KUKA KRL program: EPS_2_251455_MH52A_A_20251003061554.src

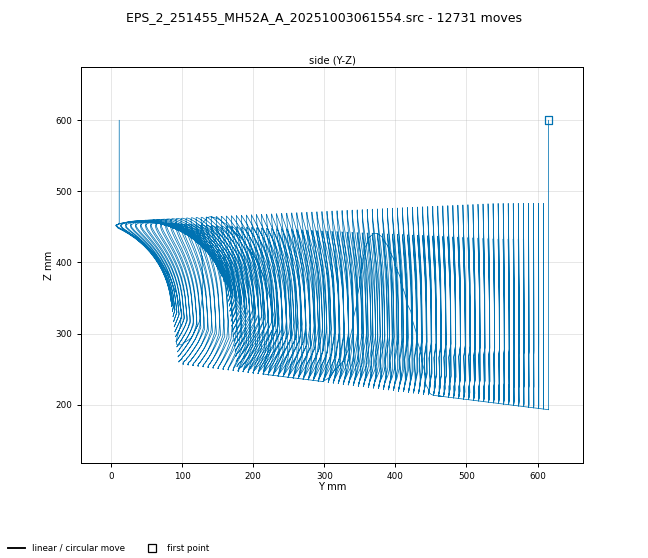
[picture p0: tool path of EPS_2_251455_MH52A_A_20251003061554.src, 12731 of 12733 moves have a stored position in this frame; points joined in program order, loops and branches not executed]
&ACCESS RVP
&REL 4
&COMMENT QRS 19112012
&PARAM EDITMASK = *
DEF PART()
EXT BAS (BAS_COMMAND :IN,REAL :IN )
INT I
BAS (#INITMOV,0 )

;KUKA QRS Post kuka4.cps  Date:22-06-2017 !

File_ID=2878

QRS_PRE_INIT()

;Init var - Until changes are made in qrs_pre_init
Outlet_Square_prg=0
Inlet_1_Square_prg=0
Inlet_2_Square_prg=0
Inlet_3_Square_prg=0
Inlet_4_Square_prg=0
Inlet_5_Square_prg=0

Outlet_1={X 0.000, Y 540.910, Z 382.500, B 0.000, E1 0.000 }
Inlet_1={X 0.000, Y 544.470, Z 332.500, B 0.000, E1 195.000 }
Outlet_1_type=201
Inlet_1_type=201
;QRS#1=Sidecore dimensions
;QRS#2=200-8" PVC SDR 35
;QRS#3=200-8" PVC SDR 35
;QRS#4=
;QRS#5=
;QRS#6=
;QRS#7=
;QRS#8=
;QRS#9=12-08 PSX
;QRS#10=12-08 PSX
;QRS#11=
;QRS#12=
;QRS#13=
;QRS#14=
;QRS#15=
;QRS#16=1220x127x762 2,5'
;QRS#17=EPS Height
;QRS#18=483
;QRS#19=*
;QRS#20= UPDATED VERSION 22-06-2017
;QRS#21=*
Outlet_Square=0100
Inlet_1_Square=0100
Inlet_2_Square=0
Inlet_3_Square=0
Inlet_4_Square=0
Inlet_5_Square=0
Mill_Square=1
Outlet_Square_Prg=204
Inlet_1_Square_prg=204

QRS_INIT()

$ADVANCE=5

; T1
PTP {E1 173.581,E2 173.581}
PTP {X 0,Y 615.464,A -85,B 0,C 180,E1 173.581,E2 173.581,E3 0,E4 0,E5 0,E6 0}
QRS_SPEED_INIT()
LIN {X 0,Y 615.464,Z 600,A -85,B 0,C 180,E1 173.581,E2 173.581,E3 0,E4 0,E5 0,E6 0} C_VEL
LIN {X 0,Y 615.464,Z 202.872,A -85,B 0,C 180,E1 173.581,E2 173.581} C_VEL
LIN {X 0,Y 615.464,Z 194.699,A -85,B 0,C 180,E1 173.581,E2 173.581} C_VEL
LIN {X 0,Y 615.452,Z 192.699,A -85,B 0,C 180,E1 173.395,E2 173.395} C_VEL
LIN {X 0,Y 615.457,Z 192.7,A -85,B 0,C 180,E1 170.801,E2 170.801} C_VEL
LIN {X 0,Y 615.41,Z 192.7,A -85,B 0,C 180,E1 168.138,E2 168.138} C_VEL
LIN {X 0,Y 615.458,Z 192.7,A -85,B 0,C 180,E1 165.45,E2 165.45} C_VEL
LIN {X 0,Y 615.437,Z 192.699,A -85,B 0,C 180,E1 162.728,E2 162.728} C_VEL
LIN {X 0,Y 615.43,Z 192.699,A -85,B 0,C 180,E1 160.66,E2 160.66} C_VEL
LIN {X 0,Y 615.423,Z 192.699,A -85,B 0,C 180,E1 158.566,E2 158.566} C_VEL
LIN {X 0,Y 615.417,Z 192.699,A -85,B 0,C 180,E1 156.441,E2 156.441} C_VEL
LIN {X 0,Y 615.416,Z 192.699,A -85,B 0,C 180,E1 154.281,E2 154.281} C_VEL
LIN {X 0,Y 615.475,Z 192.701,A -85,B 0,C 180,E1 151.54,E2 151.54} C_VEL
LIN {X 0,Y 615.443,Z 192.697,A -85,B 0,C 180,E1 148.91,E2 148.91} C_VEL
LIN {X 0,Y 615.419,Z 192.698,A -85,B 0,C 180,E1 146.465,E2 146.465} C_VEL
LIN {X 0,Y 615.429,Z 192.699,A -85,B 0,C 180,E1 144.165,E2 144.165} C_VEL
LIN {X 0,Y 615.453,Z 192.699,A -85,B 0,C 180,E1 141.929,E2 141.929} C_VEL
LIN {X 0,Y 615.488,Z 192.695,A -85,B 0,C 180,E1 139.394,E2 139.394} C_VEL
LIN {X 0,Y 615.428,Z 192.696,A -85,B 0,C 180,E1 136.75,E2 136.75} C_VEL
LIN {X 0,Y 615.461,Z 192.699,A -85,B 0,C 180,E1 133.995,E2 133.995} C_VEL
LIN {X 0,Y 615.446,Z 192.694,A -85,B 0,C 180,E1 131.09,E2 131.09} C_VEL
LIN {X 0,Y 615.432,Z 192.695,A -85,B 0,C 180,E1 128.903,E2 128.903} C_VEL
LIN {X 0,Y 615.438,Z 192.697,A -85,B 0,C 180,E1 126.423,E2 126.423} C_VEL
LIN {X 0,Y 615.476,Z 192.7,A -85,B 0,C 180,E1 124.018,E2 124.018} C_VEL
LIN {X 0,Y 615.44,Z 192.694,A -85,B 0,C 180,E1 121.079,E2 121.079} C_VEL
LIN {X 0,Y 615.437,Z 192.696,A -85,B 0,C 180,E1 118.656,E2 118.656} C_VEL
LIN {X 0,Y 615.499,Z 192.69,A -85,B 0,C 180,E1 115.711,E2 115.711} C_VEL
LIN {X 0,Y 615.475,Z 192.69,A -85,B 0,C 180,E1 113.553,E2 113.553} C_VEL
LIN {X 0,Y 615.459,Z 192.691,A -85,B 0,C 180,E1 111.43,E2 111.43} C_VEL
LIN {X 0,Y 615.451,Z 192.692,A -85,B 0,C 180,E1 109.336,E2 109.336} C_VEL
LIN {X 0,Y 615.446,Z 192.692,A -85,B 0,C 180,E1 107.269,E2 107.269} C_VEL
LIN {X 0,Y 615.444,Z 192.692,A -85,B 0,C 180,E1 105.225,E2 105.225} C_VEL
LIN {X 0,Y 615.443,Z 192.693,A -85,B 0,C 180,E1 103.2,E2 103.2} C_VEL
LIN {X 0,Y 615.47,Z 192.698,A -85,B 0,C 180,E1 100.525,E2 100.525} C_VEL
LIN {X 0,Y 615.485,Z 192.689,A -85,B 0,C 180,E1 97.874,E2 97.874} C_VEL
LIN {X 0,Y 615.444,Z 192.693,A -85,B 0,C 180,E1 95.24,E2 95.24} C_VEL
LIN {X 0,Y 615.449,Z 192.72,A -85,B 0,C 180,E1 92.985,E2 92.985} C_VEL
LIN {X 0,Y 615.487,Z 207.89,A -85,B 0,C 180,E1 90.326,E2 90.326} C_VEL
LIN {X 0,Y 615.49,Z 222.406,A -85,B 0,C 180,E1 87.811,E2 87.811} C_VEL
LIN {X 0,Y 615.462,Z 329.005,A -85,B 0,C 180,E1 86.542,E2 86.542} C_VEL
LIN {X 0,Y 615.477,Z 341.266,A -85,B 0,C 180,E1 86.276,E2 86.276} C_VEL
LIN {X 0,Y 615.495,Z 353.971,A -85,B 0,C 180,E1 85.866,E2 85.866} C_VEL
LIN {X 0,Y 615.468,Z 366.154,A -85,B 0,C 180,E1 85.333,E2 85.333} C_VEL
LIN {X 0,Y 615.471,Z 377.623,A -85,B 0,C 180,E1 84.676,E2 84.676} C_VEL
LIN {X 0,Y 615.498,Z 387.942,A -85,B 0,C 180,E1 83.937,E2 83.937} C_VEL
LIN {X 0,Y 615.497,Z 397.467,A -85,B 0,C 180,E1 83.098,E2 83.098} C_VEL
LIN {X 0,Y 615.496,Z 406.346,A -85,B 0,C 180,E1 82.124,E2 82.124} C_VEL
LIN {X 0,Y 615.496,Z 413.655,A -85,B 0,C 180,E1 81.132,E2 81.132} C_VEL
LIN {X 0,Y 615.499,Z 419.524,A -85,B 0,C 180,E1 80.138,E2 80.138} C_VEL
LIN {X 0,Y 615.494,Z 424.293,A -85,B 0,C 180,E1 79.108,E2 79.108} C_VEL
LIN {X 0,Y 615.496,Z 427.682,A -85,B 0,C 180,E1 78.139,E2 78.139} C_VEL
LIN {X 0,Y 615.495,Z 429.469,A -85,B 0,C 180,E1 77.47,E2 77.47} C_VEL
LIN {X 0,Y 615.496,Z 430.806,A -85,B 0,C 180,E1 76.799,E2 76.799} C_VEL
LIN {X 0,Y 615.498,Z 431.817,A -85,B 0,C 180,E1 76.063,E2 76.063} C_VEL
LIN {X 0,Y 615.494,Z 432.275,A -85,B 0,C 180,E1 75.451,E2 75.451} C_VEL
LIN {X 0,Y 615.496,Z 432.351,A -85,B 0,C 180,E1 74.774,E2 74.774} C_VEL
LIN {X 0,Y 615.494,Z 431.486,A -85,B 0,C 180,E1 73.566,E2 73.566} C_VEL
LIN {X 0,Y 615.495,Z 430.097,A -85,B 0,C 180,E1 72.73,E2 72.73} C_VEL
LIN {X 0,Y 615.498,Z 428.448,A -85,B 0,C 180,E1 72.044,E2 72.044} C_VEL
LIN {X 0,Y 615.496,Z 425.076,A -85,B 0,C 180,E1 71.009,E2 71.009} C_VEL
LIN {X 0,Y 615.496,Z 420.512,A -85,B 0,C 180,E1 69.968,E2 69.968} C_VEL
LIN {X 0,Y 615.496,Z 414.592,A -85,B 0,C 180,E1 68.92,E2 68.92} C_VEL
LIN {X 0,Y 615.497,Z 406.993,A -85,B 0,C 180,E1 67.865,E2 67.865} C_VEL
LIN {X 0,Y 615.498,Z 399.11,A -85,B 0,C 180,E1 66.979,E2 66.979} C_VEL
LIN {X 0,Y 615.497,Z 389.577,A -85,B 0,C 180,E1 66.103,E2 66.103} C_VEL
LIN {X 0,Y 615.48,Z 379.696,A -85,B 0,C 180,E1 65.37,E2 65.37} C_VEL
LIN {X 0,Y 615.466,Z 368.848,A -85,B 0,C 180,E1 64.72,E2 64.72} C_VEL
LIN {X 0,Y 615.483,Z 356.684,A -85,B 0,C 180,E1 64.149,E2 64.149} C_VEL
LIN {X 0,Y 615.446,Z 345.029,A -85,B 0,C 180,E1 63.738,E2 63.738} C_VEL
LIN {X 0,Y 615.434,Z 332.142,A -85,B 0,C 180,E1 63.425,E2 63.425} C_VEL
LIN {X 0,Y 615.438,Z 314.635,A -85,B 0,C 180,E1 63.184,E2 63.184} C_VEL
LIN {X 0,Y 615.475,Z 222.334,A -85,B 0,C 180,E1 62.086,E2 62.086} C_VEL
LIN {X 0,Y 615.486,Z 206.099,A -85,B 0,C 180,E1 59.272,E2 59.272} C_VEL
LIN {X 0,Y 615.471,Z 192.69,A -85,B 0,C 180,E1 56.911,E2 56.911} C_VEL
LIN {X 0,Y 615.487,Z 192.686,A -85,B 0,C 180,E1 54.166,E2 54.166} C_VEL
LIN {X 0,Y 615.486,Z 192.692,A -85,B 0,C 180,E1 51.934,E2 51.934} C_VEL
LIN {X 0,Y 615.477,Z 192.696,A -85,B 0,C 180,E1 49.396,E2 49.396} C_VEL
LIN {X 0,Y 615.476,Z 192.685,A -85,B 0,C 180,E1 46.758,E2 46.758} C_VEL
LIN {X 0,Y 615.488,Z 192.695,A -85,B 0,C 180,E1 44.001,E2 44.001} C_VEL
LIN {X 0,Y 615.469,Z 192.695,A -85,B 0,C 180,E1 41.475,E2 41.475} C_VEL
LIN {X 0,Y 615.468,Z 192.687,A -85,B 0,C 180,E1 38.906,E2 38.906} C_VEL
LIN {X 0,Y 615.488,Z 192.688,A -85,B 0,C 180,E1 36.424,E2 36.424} C_VEL
LIN {X 0,Y 615.492,Z 192.701,A -85,B 0,C 180,E1 34.021,E2 34.021} C_VEL
LIN {X 0,Y 615.466,Z 192.696,A -85,B 0,C 180,E1 31.686,E2 31.686} C_VEL
LIN {X 0,Y 615.454,Z 192.692,A -85,B 0,C 180,E1 29.408,E2 29.408} C_VEL
LIN {X 0,Y 615.465,Z 192.688,A -85,B 0,C 180,E1 27.049,E2 27.049} C_VEL
LIN {X 0,Y 615.476,Z 192.698,A -85,B 0,C 180,E1 24.015,E2 24.015} C_VEL
LIN {X 0,Y 615.449,Z 192.692,A -85,B 0,C 180,E1 21.433,E2 21.433} C_VEL
LIN {X 0,Y 615.493,Z 192.692,A -85,B 0,C 180,E1 18.618,E2 18.618} C_VEL
LIN {X 0,Y 615.452,Z 192.696,A -85,B 0,C 180,E1 15.906,E2 15.906} C_VEL
LIN {X 0,Y 615.447,Z 192.696,A -85,B 0,C 180,E1 13.875,E2 13.875} C_VEL
LIN {X 0,Y 615.444,Z 192.695,A -85,B 0,C 180,E1 11.861,E2 11.861} C_VEL
LIN {X 0,Y 615.442,Z 192.695,A -85,B 0,C 180,E1 9.863,E2 9.863} C_VEL
LIN {X 0,Y 615.439,Z 192.695,A -85,B 0,C 180,E1 7.876,E2 7.876} C_VEL
LIN {X 0,Y 615.463,Z 192.691,A -85,B 0,C 180,E1 5.241,E2 5.241} C_VEL
LIN {X 0,Y 615.484,Z 192.701,A -85,B 0,C 180,E1 2.618,E2 2.618} C_VEL
LIN {X 0,Y 615.43,Z 192.697,A -85,B 0,C 180,E1 0,E2 0} C_VEL
LIN {X 0,Y 615.431,Z 192.697,A -85,B 0,C 180,E1 -1.963,E2 -1.963} C_VEL
LIN {X 0,Y 615.429,Z 192.697,A -85,B 0,C 180,E1 -3.929,E2 -3.929} C_VEL
LIN {X 0,Y 615.428,Z 192.697,A -85,B 0,C 180,E1 -5.899,E2 -5.899} C_VEL
LIN {X 0,Y 615.423,Z 192.698,A -85,B 0,C 180,E1 -7.877,E2 -7.877} C_VEL
LIN {X 0,Y 615.424,Z 192.698,A -85,B 0,C 180,E1 -9.863,E2 -9.863} C_VEL
LIN {X 0,Y 615.421,Z 192.698,A -85,B 0,C 180,E1 -11.862,E2 -11.862} C_VEL
LIN {X 0,Y 615.458,Z 192.697,A -85,B 0,C 180,E1 -14.55,E2 -14.55} C_VEL
LIN {X 0,Y 615.445,Z 192.7,A -85,B 0,C 180,E1 -17.272,E2 -17.272} C_VEL
LIN {X 0,Y 615.433,Z 192.7,A -85,B 0,C 180,E1 -19.34,E2 -19.34} C_VEL
LIN {X 0,Y 615.422,Z 192.7,A -85,B 0,C 180,E1 -21.435,E2 -21.435} C_VEL
LIN {X 0,Y 615.411,Z 192.701,A -85,B 0,C 180,E1 -23.56,E2 -23.56} C_VEL
LIN {X 0,Y 615.412,Z 192.7,A -85,B 0,C 180,E1 -25.719,E2 -25.719} C_VEL
LIN {X 0,Y 615.47,Z 192.701,A -85,B 0,C 180,E1 -28.455,E2 -28.455} C_VEL
LIN {X 0,Y 615.443,Z 192.698,A -85,B 0,C 180,E1 -31.086,E2 -31.086} C_VEL
LIN {X 0,Y 615.419,Z 192.698,A -85,B 0,C 180,E1 -33.53,E2 -33.53} C_VEL
LIN {X 0,Y 615.429,Z 192.699,A -85,B 0,C 180,E1 -35.831,E2 -35.831} C_VEL
LIN {X 0,Y 615.454,Z 192.699,A -85,B 0,C 180,E1 -38.071,E2 -38.071} C_VEL
LIN {X 0,Y 615.486,Z 192.695,A -85,B 0,C 180,E1 -40.607,E2 -40.607} C_VEL
LIN {X 0,Y 615.43,Z 192.696,A -85,B 0,C 180,E1 -43.25,E2 -43.25} C_VEL
LIN {X 0,Y 615.467,Z 192.699,A -85,B 0,C 180,E1 -46.005,E2 -46.005} C_VEL
LIN {X 0,Y 615.448,Z 192.693,A -85,B 0,C 180,E1 -48.91,E2 -48.91} C_VEL
LIN {X 0,Y 615.435,Z 192.695,A -85,B 0,C 180,E1 -51.095,E2 -51.095} C_VEL
LIN {X 0,Y 615.444,Z 192.698,A -85,B 0,C 180,E1 -53.575,E2 -53.575} C_VEL
LIN {X 0,Y 615.486,Z 192.689,A -85,B 0,C 180,E1 -56.467,E2 -56.467} C_VEL
LIN {X 0,Y 615.442,Z 192.693,A -85,B 0,C 180,E1 -59.08,E2 -59.08} C_VEL
LIN {X 0,Y 615.458,Z 192.698,A -85,B 0,C 180,E1 -61.555,E2 -61.555} C_VEL
LIN {X 0,Y 615.48,Z 192.688,A -85,B 0,C 180,E1 -64.433,E2 -64.433} C_VEL
LIN {X 0,Y 615.447,Z 192.693,A -85,B 0,C 180,E1 -67.044,E2 -67.044} C_VEL
LIN {X 0,Y 615.482,Z 210.777,A -85,B 0,C 180,E1 -69.445,E2 -69.445} C_VEL
LIN {X 0,Y 615.489,Z 232.021,A -85,B 0,C 180,E1 -72.215,E2 -72.215} C_VEL
LIN {X 0,Y 615.494,Z 253.241,A -85,B 0,C 180,E1 -74.944,E2 -74.944} C_VEL
LIN {X 0,Y 615.452,Z 270.301,A -85,B 0,C 180,E1 -77.113,E2 -77.113} C_VEL
LIN {X 0,Y 615.478,Z 378.828,A -85,B 0,C 180,E1 -78.41,E2 -78.41} C_VEL
LIN {X 0,Y 615.47,Z 391.343,A -85,B 0,C 180,E1 -78.681,E2 -78.681} C_VEL
LIN {X 0,Y 615.486,Z 404.643,A -85,B 0,C 180,E1 -79.114,E2 -79.114} C_VEL
LIN {X 0,Y 615.483,Z 416.474,A -85,B 0,C 180,E1 -79.639,E2 -79.639} C_VEL
LIN {X 0,Y 615.495,Z 427.99,A -85,B 0,C 180,E1 -80.304,E2 -80.304} C_VEL
LIN {X 0,Y 615.499,Z 438.337,A -85,B 0,C 180,E1 -81.05,E2 -81.05} C_VEL
LIN {X 0,Y 615.497,Z 446.807,A -85,B 0,C 180,E1 -81.794,E2 -81.794} C_VEL
LIN {X 0,Y 615.498,Z 454.602,A -85,B 0,C 180,E1 -82.619,E2 -82.619} C_VEL
LIN {X 0,Y 615.496,Z 462.199,A -85,B 0,C 180,E1 -83.607,E2 -83.607} C_VEL
LIN {X 0,Y 615.498,Z 469.201,A -85,B 0,C 180,E1 -84.758,E2 -84.758} C_VEL
LIN {X 0,Y 615.494,Z 473.848,A -85,B 0,C 180,E1 -85.743,E2 -85.743} C_VEL
LIN {X 0,Y 615.494,Z 477.396,A -85,B 0,C 180,E1 -86.726,E2 -86.726} C_VEL
LIN {X 0,Y 615.497,Z 479.231,A -85,B 0,C 180,E1 -87.381,E2 -87.381} C_VEL
LIN {X 0,Y 615.499,Z 480.606,A -85,B 0,C 180,E1 -88.036,E2 -88.036} C_VEL
LIN {X 0,Y 615.496,Z 482.173,A -85,B 0,C 180,E1 -89.345,E2 -89.345} C_VEL
LIN {X 0,Y 615.494,Z 482.389,A -85,B 0,C 180,E1 -89.999,E2 -89.999} C_VEL
LIN {X 0,Y 615.495,Z 481.581,A -85,B 0,C 180,E1 -91.307,E2 -91.307} C_VEL
LIN {X 0,Y 615.499,Z 480.61,A -85,B 0,C 180,E1 -91.962,E2 -91.962} C_VEL
LIN {X 0,Y 615.497,Z 479.236,A -85,B 0,C 180,E1 -92.616,E2 -92.616} C_VEL
LIN {X 0,Y 615.496,Z 476.354,A -85,B 0,C 180,E1 -93.599,E2 -93.599} C_VEL
LIN {X 0,Y 615.498,Z 472.448,A -85,B 0,C 180,E1 -94.583,E2 -94.583} C_VEL
LIN {X 0,Y 615.499,Z 467.414,A -85,B 0,C 180,E1 -95.568,E2 -95.568} C_VEL
LIN {X 0,Y 615.496,Z 460.87,A -85,B 0,C 180,E1 -96.583,E2 -96.583} C_VEL
LIN {X 0,Y 615.497,Z 453.15,A -85,B 0,C 180,E1 -97.544,E2 -97.544} C_VEL
LIN {X 0,Y 615.498,Z 445.065,A -85,B 0,C 180,E1 -98.369,E2 -98.369} C_VEL
LIN {X 0,Y 615.499,Z 435.194,A -85,B 0,C 180,E1 -99.197,E2 -99.197} C_VEL
LIN {X 0,Y 615.492,Z 424.016,A -85,B 0,C 180,E1 -99.943,E2 -99.943} C_VEL
LIN {X 0,Y 615.485,Z 413.067,A -85,B 0,C 180,E1 -100.525,E2 -100.525} C_VEL
LIN {X 0,Y 615.476,Z 400.535,A -85,B 0,C 180,E1 -101.039,E2 -101.039} C_VEL
LIN {X 0,Y 615.471,Z 388.165,A -85,B 0,C 180,E1 -101.4,E2 -101.4} C_VEL
LIN {X 0,Y 615.481,Z 374.629,A -85,B 0,C 180,E1 -101.65,E2 -101.65} C_VEL
LIN {X 0,Y 615.452,Z 270.319,A -85,B 0,C 180,E1 -102.885,E2 -102.885} C_VEL
LIN {X 0,Y 615.487,Z 249.28,A -85,B 0,C 180,E1 -105.563,E2 -105.563} C_VEL
LIN {X 0,Y 615.456,Z 227.019,A -85,B 0,C 180,E1 -108.434,E2 -108.434} C_VEL
LIN {X 0,Y 615.482,Z 206.806,A -85,B 0,C 180,E1 -111.078,E2 -111.078} C_VEL
LIN {X 0,Y 615.447,Z 192.693,A -85,B 0,C 180,E1 -112.976,E2 -112.976} C_VEL
LIN {X 0,Y 615.499,Z 192.686,A -85,B 0,C 180,E1 -115.711,E2 -115.711} C_VEL
LIN {X 0,Y 615.451,Z 192.695,A -85,B 0,C 180,E1 -118.656,E2 -118.656} C_VEL
LIN {X 0,Y 615.447,Z 192.692,A -85,B 0,C 180,E1 -121.079,E2 -121.079} C_VEL
LIN {X 0,Y 615.496,Z 192.701,A -85,B 0,C 180,E1 -124.017,E2 -124.017} C_VEL
LIN {X 0,Y 615.454,Z 192.697,A -85,B 0,C 180,E1 -126.422,E2 -126.422} C_VEL
LIN {X 0,Y 615.445,Z 192.692,A -85,B 0,C 180,E1 -129.057,E2 -129.057} C_VEL
LIN {X 0,Y 615.487,Z 192.689,A -85,B 0,C 180,E1 -131.468,E2 -131.468} C_VEL
LIN {X 0,Y 615.465,Z 192.698,A -85,B 0,C 180,E1 -134.145,E2 -134.145} C_VEL
LIN {X 0,Y 615.436,Z 192.694,A -85,B 0,C 180,E1 -136.751,E2 -136.751} C_VEL
LIN {X 0,Y 615.489,Z 192.69,A -85,B 0,C 180,E1 -139.393,E2 -139.393} C_VEL
LIN {X 0,Y 615.467,Z 192.699,A -85,B 0,C 180,E1 -141.982,E2 -141.982} C_VEL
LIN {X 0,Y 615.435,Z 192.696,A -85,B 0,C 180,E1 -144.38,E2 -144.38} C_VEL
LIN {X 0,Y 615.437,Z 192.694,A -85,B 0,C 180,E1 -146.76,E2 -146.76} C_VEL
LIN {X 0,Y 615.465,Z 192.692,A -85,B 0,C 180,E1 -149.079,E2 -149.079} C_VEL
LIN {X 0,Y 615.441,Z 192.697,A -85,B 0,C 180,E1 -152.082,E2 -152.082} C_VEL
LIN {X 0,Y 615.428,Z 192.696,A -85,B 0,C 180,E1 -154.429,E2 -154.429} C_VEL
LIN {X 0,Y 615.484,Z 192.693,A -85,B 0,C 180,E1 -157.155,E2 -157.155} C_VEL
LIN {X 0,Y 615.438,Z 192.698,A -85,B 0,C 180,E1 -159.965,E2 -159.965} C_VEL
LIN {X 0,Y 615.431,Z 192.698,A -85,B 0,C 180,E1 -162.041,E2 -162.041} C_VEL
LIN {X 0,Y 615.425,Z 192.698,A -85,B 0,C 180,E1 -164.093,E2 -164.093} C_VEL
LIN {X 0,Y 615.424,Z 192.698,A -85,B 0,C 180,E1 -166.124,E2 -166.124} C_VEL
LIN {X 0,Y 615.423,Z 192.698,A -85,B 0,C 180,E1 -168.138,E2 -168.138} C_VEL
LIN {X 0,Y 615.419,Z 192.698,A -85,B 0,C 180,E1 -170.137,E2 -170.137} C_VEL
LIN {X 0,Y 615.458,Z 192.696,A -85,B 0,C 180,E1 -172.784,E2 -172.784} C_VEL
LIN {X 0,Y 615.462,Z 192.7,A -85,B 0,C 180,E1 -175.415,E2 -175.415} C_VEL
LIN {X 0,Y 615.417,Z 192.698,A -85,B 0,C 180,E1 -178.036,E2 -178.036} C_VEL
LIN {X 0,Y 615.452,Z 192.698,A -85,B 0,C 180,E1 -180.654,E2 -180.654} C_VEL
LIN {X 0,Y 615.462,Z 192.7,A -85,B 0,C 180,E1 -183.273,E2 -183.273} C_VEL
LIN {X 0,Y 615.412,Z 192.7,A -85,B 0,C 180,E1 -185.899,E2 -185.899} C_VEL
LIN {X 0,Y 615.452,Z 192.699,A -85,B 0,C 180,E1 -186.605,E2 -186.605} C_VEL
LIN {X 0,Y 614.783,Z 192.848,A -85,B 0,C 180,E1 -187.151,E2 -187.151} C_VEL
LIN {X 0,Y 611.954,Z 193.251,A -85,B 0,C 180,E1 -188.037,E2 -188.037} C_VEL
LIN {X 0,Y 609.556,Z 193.564,A -85,B 0,C 180,E1 -188.749,E2 -188.749} C_VEL
LIN {X 0,Y 608.507,Z 193.685,A -85,B 0,C 180,E1 -189.299,E2 -189.299} C_VEL
LIN {X 0,Y 608.411,Z 193.695,A -85,B 0,C 180,E1 -189.485,E2 -189.485} C_VEL
LIN {X 0,Y 608.428,Z 193.694,A -85,B 0,C 180,E1 -191.324,E2 -191.324} C_VEL
LIN {X 0,Y 608.405,Z 193.694,A -85,B 0,C 180,E1 -194.039,E2 -194.039} C_VEL
LIN {X 0,Y 608.437,Z 193.7,A -85,B 0,C 180,E1 -196.784,E2 -196.784} C_VEL
LIN {X 0,Y 608.392,Z 193.695,A -85,B 0,C 180,E1 -199.572,E2 -199.572} C_VEL
LIN {X 0,Y 608.408,Z 193.693,A -85,B 0,C 180,E1 -201.694,E2 -201.694} C_VEL
LIN {X 0,Y 608.416,Z 193.701,A -85,B 0,C 180,E1 -204.572,E2 -204.572} C_VEL
LIN {X 0,Y 608.395,Z 193.695,A -85,B 0,C 180,E1 -207.52,E2 -207.52} C_VEL
LIN {X 0,Y 608.412,Z 193.694,A -85,B 0,C 180,E1 -209.974,E2 -209.974} C_VEL
LIN {X 0,Y 608.451,Z 193.698,A -85,B 0,C 180,E1 -212.531,E2 -212.531} C_VEL
LIN {X 0,Y 608.397,Z 193.695,A -85,B 0,C 180,E1 -215.281,E2 -215.281} C_VEL
LIN {X 0,Y 608.425,Z 193.692,A -85,B 0,C 180,E1 -217.749,E2 -217.749} C_VEL
LIN {X 0,Y 608.441,Z 193.699,A -85,B 0,C 180,E1 -220.336,E2 -220.336} C_VEL
LIN {X 0,Y 608.412,Z 193.694,A -85,B 0,C 180,E1 -222.963,E2 -222.963} C_VEL
LIN {X 0,Y 608.407,Z 193.693,A -85,B 0,C 180,E1 -225.206,E2 -225.206} C_VEL
LIN {X 0,Y 608.434,Z 193.695,A -85,B 0,C 180,E1 -227.943,E2 -227.943} C_VEL
LIN {X 0,Y 608.446,Z 193.691,A -85,B 0,C 180,E1 -230.705,E2 -230.705} C_VEL
LIN {X 0,Y 608.405,Z 193.693,A -85,B 0,C 180,E1 -233.087,E2 -233.087} C_VEL
LIN {X 0,Y 608.43,Z 193.692,A -85,B 0,C 180,E1 -235.533,E2 -235.533} C_VEL
LIN {X 0,Y 608.444,Z 193.696,A -85,B 0,C 180,E1 -237.909,E2 -237.909} C_VEL
LIN {X 0,Y 608.479,Z 193.692,A -85,B 0,C 180,E1 -240.225,E2 -240.225} C_VEL
LIN {X 0,Y 608.407,Z 193.694,A -85,B 0,C 180,E1 -243.228,E2 -243.228} C_VEL
LIN {X 0,Y 608.48,Z 193.693,A -85,B 0,C 180,E1 -245.847,E2 -245.847} C_VEL
LIN {X 0,Y 608.455,Z 193.691,A -85,B 0,C 180,E1 -248.311,E2 -248.311} C_VEL
LIN {X 0,Y 608.429,Z 193.691,A -85,B 0,C 180,E1 -251.133,E2 -251.133} C_VEL
LIN {X 0,Y 608.457,Z 193.696,A -85,B 0,C 180,E1 -253.909,E2 -253.909} C_VEL
LIN {X 0,Y 608.435,Z 193.69,A -85,B 0,C 180,E1 -256.645,E2 -256.645} C_VEL
LIN {X 0,Y 608.441,Z 193.693,A -85,B 0,C 180,E1 -259.352,E2 -259.352} C_VEL
LIN {X 0,Y 608.475,Z 193.689,A -85,B 0,C 180,E1 -262.035,E2 -262.035} C_VEL
LIN {X 0,Y 608.43,Z 193.69,A -85,B 0,C 180,E1 -264.699,E2 -264.699} C_VEL
LIN {X 0,Y 608.44,Z 193.816,A -85,B 0,C 180,E1 -266.98,E2 -266.98} C_VEL
LIN {X 0,Y 608.486,Z 207.153,A -85,B 0,C 180,E1 -269.339,E2 -269.339} C_VEL
LIN {X 0,Y 608.499,Z 222.784,A -85,B 0,C 180,E1 -272.049,E2 -272.049} C_VEL
LIN {X 0,Y 608.52,Z 329.538,A -85,B 0,C 180,E1 -273.332,E2 -273.332} C_VEL
LIN {X 0,Y 608.518,Z 343.159,A -85,B 0,C 180,E1 -273.643,E2 -273.643} C_VEL
LIN {X 0,Y 608.535,Z 355.415,A -85,B 0,C 180,E1 -274.057,E2 -274.057} C_VEL
LIN {X 0,Y 608.474,Z 366.473,A -85,B 0,C 180,E1 -274.555,E2 -274.555} C_VEL
LIN {X 0,Y 608.457,Z 377.952,A -85,B 0,C 180,E1 -275.22,E2 -275.22} C_VEL
LIN {X 0,Y 608.498,Z 388.292,A -85,B 0,C 180,E1 -275.967,E2 -275.967} C_VEL
LIN {X 0,Y 608.46,Z 397.701,A -85,B 0,C 180,E1 -276.8,E2 -276.8} C_VEL
LIN {X 0,Y 608.454,Z 406.781,A -85,B 0,C 180,E1 -277.801,E2 -277.801} C_VEL
LIN {X 0,Y 608.449,Z 414.134,A -85,B 0,C 180,E1 -278.804,E2 -278.804} C_VEL
LIN {X 0,Y 608.433,Z 419.13,A -85,B 0,C 180,E1 -279.642,E2 -279.642} C_VEL
LIN {X 0,Y 608.436,Z 423.991,A -85,B 0,C 180,E1 -280.651,E2 -280.651} C_VEL
LIN {X 0,Y 608.434,Z 427.727,A -85,B 0,C 180,E1 -281.662,E2 -281.662} C_VEL
LIN {X 0,Y 608.419,Z 430.432,A -85,B 0,C 180,E1 -282.678,E2 -282.678} C_VEL
LIN {X 0,Y 608.439,Z 431.696,A -85,B 0,C 180,E1 -283.357,E2 -283.357} C_VEL
LIN {X 0,Y 608.422,Z 432.54,A -85,B 0,C 180,E1 -284.038,E2 -284.038} C_VEL
LIN {X 0,Y 608.416,Z 432.93,A -85,B 0,C 180,E1 -284.722,E2 -284.722} C_VEL
LIN {X 0,Y 608.418,Z 432.921,A -85,B 0,C 180,E1 -285.407,E2 -285.407} C_VEL
LIN {X 0,Y 608.422,Z 432.012,A -85,B 0,C 180,E1 -286.515,E2 -286.515} C_VEL
LIN {X 0,Y 608.42,Z 430.291,A -85,B 0,C 180,E1 -287.477,E2 -287.477} C_VEL
LIN {X 0,Y 608.427,Z 426.84,A -85,B 0,C 180,E1 -288.704,E2 -288.704} C_VEL
LIN {X 0,Y 608.428,Z 423.43,A -85,B 0,C 180,E1 -289.571,E2 -289.571} C_VEL
LIN {X 0,Y 608.435,Z 417.914,A -85,B 0,C 180,E1 -290.671,E2 -290.671} C_VEL
LIN {X 0,Y 608.464,Z 411.374,A -85,B 0,C 180,E1 -291.691,E2 -291.691} C_VEL
LIN {X 0,Y 608.466,Z 402.723,A -85,B 0,C 180,E1 -292.763,E2 -292.763} C_VEL
LIN {X 0,Y 608.472,Z 393.739,A -85,B 0,C 180,E1 -293.663,E2 -293.663} C_VEL
LIN {X 0,Y 608.479,Z 384.272,A -85,B 0,C 180,E1 -294.433,E2 -294.433} C_VEL
LIN {X 0,Y 608.458,Z 372.458,A -85,B 0,C 180,E1 -295.208,E2 -295.208} C_VEL
LIN {X 0,Y 608.528,Z 361.266,A -85,B 0,C 180,E1 -295.785,E2 -295.785} C_VEL
LIN {X 0,Y 608.483,Z 349.127,A -85,B 0,C 180,E1 -296.263,E2 -296.263} C_VEL
LIN {X 0,Y 608.487,Z 335.901,A -85,B 0,C 180,E1 -296.632,E2 -296.632} C_VEL
LIN {X 0,Y 608.503,Z 323.683,A -85,B 0,C 180,E1 -296.845,E2 -296.845} C_VEL
LIN {X 0,Y 608.477,Z 222.847,A -85,B 0,C 180,E1 -298.041,E2 -298.041} C_VEL
LIN {X 0,Y 608.474,Z 207.303,A -85,B 0,C 180,E1 -300.725,E2 -300.725} C_VEL
LIN {X 0,Y 608.452,Z 193.69,A -85,B 0,C 180,E1 -303.149,E2 -303.149} C_VEL
LIN {X 0,Y 608.47,Z 193.69,A -85,B 0,C 180,E1 -306.049,E2 -306.049} C_VEL
LIN {X 0,Y 608.456,Z 193.694,A -85,B 0,C 180,E1 -308.586,E2 -308.586} C_VEL
LIN {X 0,Y 608.456,Z 193.687,A -85,B 0,C 180,E1 -311.342,E2 -311.342} C_VEL
LIN {X 0,Y 608.457,Z 193.698,A -85,B 0,C 180,E1 -314.264,E2 -314.264} C_VEL
LIN {X 0,Y 608.434,Z 193.69,A -85,B 0,C 180,E1 -317.039,E2 -317.039} C_VEL
LIN {X 0,Y 608.455,Z 193.691,A -85,B 0,C 180,E1 -319.697,E2 -319.697} C_VEL
LIN {X 0,Y 608.459,Z 193.694,A -85,B 0,C 180,E1 -322.253,E2 -322.253} C_VEL
LIN {X 0,Y 608.464,Z 193.686,A -85,B 0,C 180,E1 -325.087,E2 -325.087} C_VEL
LIN {X 0,Y 608.461,Z 193.696,A -85,B 0,C 180,E1 -327.906,E2 -327.906} C_VEL
LIN {X 0,Y 608.453,Z 193.692,A -85,B 0,C 180,E1 -330.22,E2 -330.22} C_VEL
LIN {X 0,Y 608.452,Z 193.688,A -85,B 0,C 180,E1 -332.79,E2 -332.79} C_VEL
LIN {X 0,Y 608.469,Z 193.695,A -85,B 0,C 180,E1 -335.84,E2 -335.84} C_VEL
LIN {X 0,Y 608.443,Z 193.69,A -85,B 0,C 180,E1 -338.308,E2 -338.308} C_VEL
LIN {X 0,Y 608.459,Z 193.689,A -85,B 0,C 180,E1 -341.131,E2 -341.131} C_VEL
LIN {X 0,Y 608.44,Z 193.694,A -85,B 0,C 180,E1 -343.906,E2 -343.906} C_VEL
LIN {X 0,Y 608.435,Z 193.693,A -85,B 0,C 180,E1 -345.98,E2 -345.98} C_VEL
LIN {X 0,Y 608.445,Z 193.689,A -85,B 0,C 180,E1 -348.676,E2 -348.676} C_VEL
LIN {X 0,Y 608.451,Z 193.697,A -85,B 0,C 180,E1 -351.364,E2 -351.364} C_VEL
LIN {X 0,Y 608.417,Z 193.693,A -85,B 0,C 180,E1 -354.033,E2 -354.033} C_VEL
LIN {X 0,Y 608.452,Z 193.689,A -85,B 0,C 180,E1 -356.689,E2 -356.689} C_VEL
LIN {X 0,Y 608.474,Z 193.694,A -85,B 0,C 180,E1 -359.338,E2 -359.338} C_VEL
LIN {X 0,Y 608.402,Z 193.694,A -85,B 0,C 180,E1 -361.986,E2 -361.986} C_VEL
LIN {X 0,Y 608.399,Z 193.694,A -85,B 0,C 180,E1 -363.975,E2 -363.975} C_VEL
LIN {X 0,Y 608.437,Z 193.692,A -85,B 0,C 180,E1 -366.633,E2 -366.633} C_VEL
LIN {X 0,Y 608.448,Z 193.694,A -85,B 0,C 180,E1 -369.306,E2 -369.306} C_VEL
LIN {X 0,Y 608.448,Z 193.693,A -85,B 0,C 180,E1 -371.325,E2 -371.325} C_VEL
LIN {X 0,Y 608.406,Z 193.693,A -85,B 0,C 180,E1 -374.039,E2 -374.039} C_VEL
LIN {X 0,Y 608.445,Z 193.697,A -85,B 0,C 180,E1 -376.784,E2 -376.784} C_VEL
LIN {X 0,Y 608.395,Z 193.695,A -85,B 0,C 180,E1 -379.573,E2 -379.573} C_VEL
LIN {X 0,Y 608.408,Z 193.693,A -85,B 0,C 180,E1 -381.694,E2 -381.694} C_VEL
LIN {X 0,Y 608.414,Z 193.7,A -85,B 0,C 180,E1 -384.573,E2 -384.573} C_VEL
LIN {X 0,Y 608.397,Z 193.694,A -85,B 0,C 180,E1 -387.521,E2 -387.521} C_VEL
LIN {X 0,Y 608.411,Z 193.694,A -85,B 0,C 180,E1 -389.969,E2 -389.969} C_VEL
LIN {X 0,Y 608.425,Z 193.696,A -85,B 0,C 180,E1 -392.882,E2 -392.882} C_VEL
LIN {X 0,Y 608.398,Z 193.695,A -85,B 0,C 180,E1 -395.281,E2 -395.281} C_VEL
LIN {X 0,Y 608.428,Z 193.692,A -85,B 0,C 180,E1 -397.75,E2 -397.75} C_VEL
LIN {X 0,Y 608.462,Z 193.697,A -85,B 0,C 180,E1 -400.335,E2 -400.335} C_VEL
LIN {X 0,Y 608.414,Z 193.694,A -85,B 0,C 180,E1 -402.964,E2 -402.964} C_VEL
LIN {X 0,Y 608.412,Z 193.693,A -85,B 0,C 180,E1 -405.204,E2 -405.204} C_VEL
LIN {X 0,Y 608.443,Z 193.695,A -85,B 0,C 180,E1 -407.94,E2 -407.94} C_VEL
LIN {X 0,Y 608.421,Z 193.693,A -85,B 0,C 180,E1 -410.709,E2 -410.709} C_VEL
LIN {X 0,Y 608.409,Z 193.693,A -85,B 0,C 180,E1 -413.084,E2 -413.084} C_VEL
LIN {X 0,Y 608.44,Z 193.692,A -85,B 0,C 180,E1 -415.531,E2 -415.531} C_VEL
LIN {X 0,Y 608.453,Z 193.697,A -85,B 0,C 180,E1 -417.907,E2 -417.907} C_VEL
LIN {X 0,Y 608.479,Z 193.69,A -85,B 0,C 180,E1 -420.223,E2 -420.223} C_VEL
LIN {X 0,Y 608.418,Z 193.693,A -85,B 0,C 180,E1 -423.226,E2 -423.226} C_VEL
LIN {X 0,Y 608.484,Z 193.694,A -85,B 0,C 180,E1 -425.847,E2 -425.847} C_VEL
LIN {X 0,Y 608.449,Z 193.828,A -85,B 0,C 180,E1 -426.922,E2 -426.922} C_VEL
LIN {X 0,Y 608.557,Z 208.119,A -85,B 0,C 180,E1 -428.846,E2 -428.846} C_VEL
LIN {X 0,Y 608.5,Z 228.263,A -85,B 0,C 180,E1 -431.508,E2 -431.508} C_VEL
LIN {X 0,Y 608.5,Z 249.333,A -85,B 0,C 180,E1 -434.252,E2 -434.252} C_VEL
LIN {X 0,Y 608.45,Z 270.522,A -85,B 0,C 180,E1 -436.973,E2 -436.973} C_VEL
LIN {X 0,Y 608.539,Z 378.942,A -85,B 0,C 180,E1 -438.276,E2 -438.276} C_VEL
LIN {X 0,Y 608.505,Z 392.212,A -85,B 0,C 180,E1 -438.571,E2 -438.571} C_VEL
LIN {X 0,Y 608.513,Z 404.639,A -85,B 0,C 180,E1 -438.983,E2 -438.983} C_VEL
LIN {X 0,Y 608.504,Z 416.631,A -85,B 0,C 180,E1 -439.519,E2 -439.519} C_VEL
LIN {X 0,Y 608.486,Z 428.193,A -85,B 0,C 180,E1 -440.191,E2 -440.191} C_VEL
LIN {X 0,Y 608.485,Z 438.59,A -85,B 0,C 180,E1 -440.945,E2 -440.945} C_VEL
LIN {X 0,Y 608.475,Z 447.108,A -85,B 0,C 180,E1 -441.698,E2 -441.698} C_VEL
LIN {X 0,Y 608.471,Z 454.956,A -85,B 0,C 180,E1 -442.533,E2 -442.533} C_VEL
LIN {X 0,Y 608.461,Z 462.285,A -85,B 0,C 180,E1 -443.484,E2 -443.484} C_VEL
LIN {X 0,Y 608.45,Z 467.862,A -85,B 0,C 180,E1 -444.365,E2 -444.365} C_VEL
LIN {X 0,Y 608.432,Z 472.947,A -85,B 0,C 180,E1 -445.361,E2 -445.361} C_VEL
LIN {X 0,Y 608.449,Z 476.893,A -85,B 0,C 180,E1 -446.357,E2 -446.357} C_VEL
LIN {X 0,Y 608.425,Z 479.807,A -85,B 0,C 180,E1 -447.351,E2 -447.351} C_VEL
LIN {X 0,Y 608.444,Z 481.2,A -85,B 0,C 180,E1 -448.013,E2 -448.013} C_VEL
LIN {X 0,Y 608.438,Z 482.783,A -85,B 0,C 180,E1 -449.337,E2 -449.337} C_VEL
LIN {X 0,Y 608.434,Z 483,A -85,B 0,C 180,E1 -449.999,E2 -449.999} C_VEL
LIN {X 0,Y 608.448,Z 482.185,A -85,B 0,C 180,E1 -451.322,E2 -451.322} C_VEL
LIN {X 0,Y 608.444,Z 481.204,A -85,B 0,C 180,E1 -451.984,E2 -451.984} C_VEL
LIN {X 0,Y 608.425,Z 479.813,A -85,B 0,C 180,E1 -452.647,E2 -452.647} C_VEL
LIN {X 0,Y 608.449,Z 476.901,A -85,B 0,C 180,E1 -453.641,E2 -453.641} C_VEL
LIN {X 0,Y 608.432,Z 472.957,A -85,B 0,C 180,E1 -454.636,E2 -454.636} C_VEL
LIN {X 0,Y 608.437,Z 466.887,A -85,B 0,C 180,E1 -455.799,E2 -455.799} C_VEL
LIN {X 0,Y 608.461,Z 460.248,A -85,B 0,C 180,E1 -456.798,E2 -456.798} C_VEL
LIN {X 0,Y 608.455,Z 452.006,A -85,B 0,C 180,E1 -457.798,E2 -457.798} C_VEL
LIN {X 0,Y 608.472,Z 443.559,A -85,B 0,C 180,E1 -458.634,E2 -458.634} C_VEL
LIN {X 0,Y 608.479,Z 433.119,A -85,B 0,C 180,E1 -459.471,E2 -459.471} C_VEL
LIN {X 0,Y 608.496,Z 422.791,A -85,B 0,C 180,E1 -460.143,E2 -460.143} C_VEL
LIN {X 0,Y 608.519,Z 411.307,A -85,B 0,C 180,E1 -460.738,E2 -460.738} C_VEL
LIN {X 0,Y 608.523,Z 398.949,A -85,B 0,C 180,E1 -461.223,E2 -461.223} C_VEL
LIN {X 0,Y 608.535,Z 385.536,A -85,B 0,C 180,E1 -461.595,E2 -461.595} C_VEL
LIN {X 0,Y 608.547,Z 373.255,A -85,B 0,C 180,E1 -461.806,E2 -461.806} C_VEL
LIN {X 0,Y 608.438,Z 270.457,A -85,B 0,C 180,E1 -463.036,E2 -463.036} C_VEL
LIN {X 0,Y 608.5,Z 249.352,A -85,B 0,C 180,E1 -465.746,E2 -465.746} C_VEL
LIN {X 0,Y 608.5,Z 228.273,A -85,B 0,C 180,E1 -468.491,E2 -468.491} C_VEL
LIN {X 0,Y 608.557,Z 208.138,A -85,B 0,C 180,E1 -471.152,E2 -471.152} C_VEL
LIN {X 0,Y 608.446,Z 193.763,A -85,B 0,C 180,E1 -473.087,E2 -473.087} C_VEL
LIN {X 0,Y 608.474,Z 193.688,A -85,B 0,C 180,E1 -475.721,E2 -475.721} C_VEL
LIN {X 0,Y 608.446,Z 193.691,A -85,B 0,C 180,E1 -478.615,E2 -478.615} C_VEL
LIN {X 0,Y 608.45,Z 193.691,A -85,B 0,C 180,E1 -480.542,E2 -480.542} C_VEL
LIN {X 0,Y 608.431,Z 193.69,A -85,B 0,C 180,E1 -482.876,E2 -482.876} C_VEL
LIN {X 0,Y 608.431,Z 193.691,A -85,B 0,C 180,E1 -485.273,E2 -485.273} C_VEL
LIN {X 0,Y 608.452,Z 193.693,A -85,B 0,C 180,E1 -488.238,E2 -488.238} C_VEL
LIN {X 0,Y 608.427,Z 193.695,A -85,B 0,C 180,E1 -490.326,E2 -490.326} C_VEL
LIN {X 0,Y 608.416,Z 193.692,A -85,B 0,C 180,E1 -492.957,E2 -492.957} C_VEL
LIN {X 0,Y 608.454,Z 193.696,A -85,B 0,C 180,E1 -495.729,E2 -495.729} C_VEL
LIN {X 0,Y 608.46,Z 193.695,A -85,B 0,C 180,E1 -497.938,E2 -497.938} C_VEL
LIN {X 0,Y 608.434,Z 193.69,A -85,B 0,C 180,E1 -500.698,E2 -500.698} C_VEL
LIN {X 0,Y 608.429,Z 193.692,A -85,B 0,C 180,E1 -503.083,E2 -503.083} C_VEL
LIN {X 0,Y 608.456,Z 193.695,A -85,B 0,C 180,E1 -505.53,E2 -505.53} C_VEL
LIN {X 0,Y 608.449,Z 193.693,A -85,B 0,C 180,E1 -507.904,E2 -507.904} C_VEL
LIN {X 0,Y 608.421,Z 193.693,A -85,B 0,C 180,E1 -510.218,E2 -510.218} C_VEL
LIN {X 0,Y 608.437,Z 193.69,A -85,B 0,C 180,E1 -512.788,E2 -512.788} C_VEL
LIN {X 0,Y 608.439,Z 193.694,A -85,B 0,C 180,E1 -515.841,E2 -515.841} C_VEL
LIN {X 0,Y 608.42,Z 193.692,A -85,B 0,C 180,E1 -518.306,E2 -518.306} C_VEL
LIN {X 0,Y 608.402,Z 193.694,A -85,B 0,C 180,E1 -520.428,E2 -520.428} C_VEL
LIN {X 0,Y 608.467,Z 193.695,A -85,B 0,C 180,E1 -523.45,E2 -523.45} C_VEL
LIN {X 0,Y 608.412,Z 193.694,A -85,B 0,C 180,E1 -525.979,E2 -525.979} C_VEL
LIN {X 0,Y 608.408,Z 193.694,A -85,B 0,C 180,E1 -527.999,E2 -527.999} C_VEL
LIN {X 0,Y 608.397,Z 193.695,A -85,B 0,C 180,E1 -530.022,E2 -530.022} C_VEL
LIN {X 0,Y 608.44,Z 193.692,A -85,B 0,C 180,E1 -532.7,E2 -532.7} C_VEL
LIN {X 0,Y 608.43,Z 193.697,A -85,B 0,C 180,E1 -535.362,E2 -535.362} C_VEL
LIN {X 0,Y 608.389,Z 193.695,A -85,B 0,C 180,E1 -538.014,E2 -538.014} C_VEL
LIN {X 0,Y 608.443,Z 193.693,A -85,B 0,C 180,E1 -540.662,E2 -540.662} C_VEL
LIN {X 0,Y 608.449,Z 193.693,A -85,B 0,C 180,E1 -543.311,E2 -543.311} C_VEL
LIN {X 0,Y 608.39,Z 193.695,A -85,B 0,C 180,E1 -545.967,E2 -545.967} C_VEL
LIN {X 0,Y 608.407,Z 193.693,A -85,B 0,C 180,E1 -547.968,E2 -547.968} C_VEL
LIN {X 0,Y 608.411,Z 193.695,A -85,B 0,C 180,E1 -549.485,E2 -549.485} C_VEL
LIN {X 0,Y 607.714,Z 193.782,A -85,B 0,C 180,E1 -550.038,E2 -550.038} C_VEL
LIN {X 0,Y 604.848,Z 194.146,A -85,B 0,C 180,E1 -550.935,E2 -550.935} C_VEL
LIN {X 0,Y 602.451,Z 194.439,A -85,B 0,C 180,E1 -551.657,E2 -551.657} C_VEL
LIN {X 0,Y 601.434,Z 194.563,A -85,B 0,C 180,E1 -552.214,E2 -552.214} C_VEL
LIN {X 0,Y 601.356,Z 194.575,A -85,B 0,C 180,E1 -552.402,E2 -552.402} C_VEL
LIN {X 0,Y 601.386,Z 194.577,A -85,B 0,C 180,E1 -554.898,E2 -554.898} C_VEL
LIN {X 0,Y 601.385,Z 194.575,A -85,B 0,C 180,E1 -556.987,E2 -556.987} C_VEL
LIN {X 0,Y 601.352,Z 194.572,A -85,B 0,C 180,E1 -559.811,E2 -559.811} C_VEL
LIN {X 0,Y 601.363,Z 194.571,A -85,B 0,C 180,E1 -561.961,E2 -561.961} C_VEL
LIN {X 0,Y 601.384,Z 194.572,A -85,B 0,C 180,E1 -564.296,E2 -564.296} C_VEL
LIN {X 0,Y 601.408,Z 194.568,A -85,B 0,C 180,E1 -567.113,E2 -567.113} C_VEL
LIN {X 0,Y 601.369,Z 194.57,A -85,B 0,C 180,E1 -569.396,E2 -569.396} C_VEL
LIN {X 0,Y 601.371,Z 194.57,A -85,B 0,C 180,E1 -571.728,E2 -571.728} C_VEL
LIN {X 0,Y 601.383,Z 194.572,A -85,B 0,C 180,E1 -574.121,E2 -574.121} C_VEL
LIN {X 0,Y 601.376,Z 194.577,A -85,B 0,C 180,E1 -576.585,E2 -576.585} C_VEL
LIN {X 0,Y 601.368,Z 194.571,A -85,B 0,C 180,E1 -579.13,E2 -579.13} C_VEL
LIN {X 0,Y 601.386,Z 194.569,A -85,B 0,C 180,E1 -581.768,E2 -581.768} C_VEL
LIN {X 0,Y 601.387,Z 194.574,A -85,B 0,C 180,E1 -584.539,E2 -584.539} C_VEL
LIN {X 0,Y 601.37,Z 194.57,A -85,B 0,C 180,E1 -587.333,E2 -587.333} C_VEL
LIN {X 0,Y 601.383,Z 194.575,A -85,B 0,C 180,E1 -590.009,E2 -590.009} C_VEL
LIN {X 0,Y 601.406,Z 194.569,A -85,B 0,C 180,E1 -592.621,E2 -592.621} C_VEL
LIN {X 0,Y 601.37,Z 194.57,A -85,B 0,C 180,E1 -595.07,E2 -595.07} C_VEL
LIN {X 0,Y 601.39,Z 194.569,A -85,B 0,C 180,E1 -597.487,E2 -597.487} C_VEL
LIN {X 0,Y 601.43,Z 194.569,A -85,B 0,C 180,E1 -599.851,E2 -599.851} C_VEL
LIN {X 0,Y 601.395,Z 194.567,A -85,B 0,C 180,E1 -602.89,E2 -602.89} C_VEL
LIN {X 0,Y 601.43,Z 194.568,A -85,B 0,C 180,E1 -605.708,E2 -605.708} C_VEL
LIN {X 0,Y 601.396,Z 194.575,A -85,B 0,C 180,E1 -608.044,E2 -608.044} C_VEL
LIN {X 0,Y 601.398,Z 194.566,A -85,B 0,C 180,E1 -610.903,E2 -610.903} C_VEL
LIN {X 0,Y 601.419,Z 194.572,A -85,B 0,C 180,E1 -613.715,E2 -613.715} C_VEL
LIN {X 0,Y 601.397,Z 194.567,A -85,B 0,C 180,E1 -616.486,E2 -616.486} C_VEL
LIN {X 0,Y 601.383,Z 194.571,A -85,B 0,C 180,E1 -619.225,E2 -619.225} C_VEL
LIN {X 0,Y 601.436,Z 194.568,A -85,B 0,C 180,E1 -621.941,E2 -621.941} C_VEL
LIN {X 0,Y 601.401,Z 194.566,A -85,B 0,C 180,E1 -624.637,E2 -624.637} C_VEL
LIN {X 0,Y 601.401,Z 194.601,A -85,B 0,C 180,E1 -626.903,E2 -626.903} C_VEL
LIN {X 0,Y 601.456,Z 208.169,A -85,B 0,C 180,E1 -629.332,E2 -629.332} C_VEL
LIN {X 0,Y 601.415,Z 222.621,A -85,B 0,C 180,E1 -631.884,E2 -631.884} C_VEL
LIN {X 0,Y 601.671,Z 228.51,A -85,B 0,C 180,E1 -631.967,E2 -631.967} C_VEL
LIN {X 0,Y 601.577,Z 328.847,A -85,B 0,C 180,E1 -633.182,E2 -633.182} C_VEL
LIN {X 0,Y 601.555,Z 341.965,A -85,B 0,C 180,E1 -633.475,E2 -633.475} C_VEL
LIN {X 0,Y 601.543,Z 354.546,A -85,B 0,C 180,E1 -633.895,E2 -633.895} C_VEL
LIN {X 0,Y 601.496,Z 366.628,A -85,B 0,C 180,E1 -634.44,E2 -634.44} C_VEL
LIN {X 0,Y 601.441,Z 378.086,A -85,B 0,C 180,E1 -635.113,E2 -635.113} C_VEL
LIN {X 0,Y 601.465,Z 388.404,A -85,B 0,C 180,E1 -635.869,E2 -635.869} C_VEL
LIN {X 0,Y 601.41,Z 397.789,A -85,B 0,C 180,E1 -636.711,E2 -636.711} C_VEL
LIN {X 0,Y 601.394,Z 406.852,A -85,B 0,C 180,E1 -637.724,E2 -637.724} C_VEL
LIN {X 0,Y 601.383,Z 414.191,A -85,B 0,C 180,E1 -638.739,E2 -638.739} C_VEL
LIN {X 0,Y 601.344,Z 420.093,A -85,B 0,C 180,E1 -639.757,E2 -639.757} C_VEL
LIN {X 0,Y 601.353,Z 425.504,A -85,B 0,C 180,E1 -640.977,E2 -640.977} C_VEL
LIN {X 0,Y 601.342,Z 429.227,A -85,B 0,C 180,E1 -642.144,E2 -642.144} C_VEL
LIN {X 0,Y 601.325,Z 430.817,A -85,B 0,C 180,E1 -642.83,E2 -642.83} C_VEL
LIN {X 0,Y 601.348,Z 432.567,A -85,B 0,C 180,E1 -644.064,E2 -644.064} C_VEL
LIN {X 0,Y 601.313,Z 432.972,A -85,B 0,C 180,E1 -644.9,E2 -644.9} C_VEL
LIN {X 0,Y 601.324,Z 432.866,A -85,B 0,C 180,E1 -645.593,E2 -645.593} C_VEL
LIN {X 0,Y 601.322,Z 431.944,A -85,B 0,C 180,E1 -646.589,E2 -646.589} C_VEL
LIN {X 0,Y 601.319,Z 429.892,A -85,B 0,C 180,E1 -647.69,E2 -647.69} C_VEL
LIN {X 0,Y 601.343,Z 426.661,A -85,B 0,C 180,E1 -648.798,E2 -648.798} C_VEL
LIN {X 0,Y 601.336,Z 422.624,A -85,B 0,C 180,E1 -649.811,E2 -649.811} C_VEL
LIN {X 0,Y 601.379,Z 416.678,A -85,B 0,C 180,E1 -650.947,E2 -650.947} C_VEL
LIN {X 0,Y 601.377,Z 409.98,A -85,B 0,C 180,E1 -651.96,E2 -651.96} C_VEL
LIN {X 0,Y 601.402,Z 402.635,A -85,B 0,C 180,E1 -652.864,E2 -652.864} C_VEL
LIN {X 0,Y 601.455,Z 393.64,A -85,B 0,C 180,E1 -653.773,E2 -653.773} C_VEL
LIN {X 0,Y 601.457,Z 383.087,A -85,B 0,C 180,E1 -654.63,E2 -654.63} C_VEL
LIN {X 0,Y 601.45,Z 372.298,A -85,B 0,C 180,E1 -655.337,E2 -655.337} C_VEL
LIN {X 0,Y 601.545,Z 360.454,A -85,B 0,C 180,E1 -655.947,E2 -655.947} C_VEL
LIN {X 0,Y 601.532,Z 347.444,A -85,B 0,C 180,E1 -656.45,E2 -656.45} C_VEL
LIN {X 0,Y 601.544,Z 334.517,A -85,B 0,C 180,E1 -656.8,E2 -656.8} C_VEL
LIN {X 0,Y 601.552,Z 321.537,A -85,B 0,C 180,E1 -657.011,E2 -657.011} C_VEL
LIN {X 0,Y 601.549,Z 223.772,A -85,B 0,C 180,E1 -658.182,E2 -658.182} C_VEL
LIN {X 0,Y 601.393,Z 222.661,A -85,B 0,C 180,E1 -658.199,E2 -658.199} C_VEL
LIN {X 0,Y 601.475,Z 207.161,A -85,B 0,C 180,E1 -660.937,E2 -660.937} C_VEL
LIN {X 0,Y 601.443,Z 194.563,A -85,B 0,C 180,E1 -663.221,E2 -663.221} C_VEL
LIN {X 0,Y 601.434,Z 194.57,A -85,B 0,C 180,E1 -666.265,E2 -666.265} C_VEL
LIN {X 0,Y 601.421,Z 194.564,A -85,B 0,C 180,E1 -669.123,E2 -669.123} C_VEL
LIN {X 0,Y 601.418,Z 194.566,A -85,B 0,C 180,E1 -671.762,E2 -671.762} C_VEL
LIN {X 0,Y 601.405,Z 194.571,A -85,B 0,C 180,E1 -674.534,E2 -674.534} C_VEL
LIN {X 0,Y 601.423,Z 194.564,A -85,B 0,C 180,E1 -677.404,E2 -677.404} C_VEL
LIN {X 0,Y 601.424,Z 194.568,A -85,B 0,C 180,E1 -680.462,E2 -680.462} C_VEL
LIN {X 0,Y 601.396,Z 194.568,A -85,B 0,C 180,E1 -683.417,E2 -683.417} C_VEL
LIN {X 0,Y 601.416,Z 194.574,A -85,B 0,C 180,E1 -686.061,E2 -686.061} C_VEL
LIN {X 0,Y 601.416,Z 194.566,A -85,B 0,C 180,E1 -688.54,E2 -688.54} C_VEL
LIN {X 0,Y 601.429,Z 194.565,A -85,B 0,C 180,E1 -691.373,E2 -691.373} C_VEL
LIN {X 0,Y 601.39,Z 194.572,A -85,B 0,C 180,E1 -694.129,E2 -694.129} C_VEL
LIN {X 0,Y 601.401,Z 194.566,A -85,B 0,C 180,E1 -696.589,E2 -696.589} C_VEL
LIN {X 0,Y 601.426,Z 194.569,A -85,B 0,C 180,E1 -699.478,E2 -699.478} C_VEL
LIN {X 0,Y 601.371,Z 194.571,A -85,B 0,C 180,E1 -702.311,E2 -702.311} C_VEL
LIN {X 0,Y 601.387,Z 194.568,A -85,B 0,C 180,E1 -704.408,E2 -704.408} C_VEL
LIN {X 0,Y 601.408,Z 194.569,A -85,B 0,C 180,E1 -707.172,E2 -707.172} C_VEL
LIN {X 0,Y 601.404,Z 194.569,A -85,B 0,C 180,E1 -709.905,E2 -709.905} C_VEL
LIN {X 0,Y 601.419,Z 194.564,A -85,B 0,C 180,E1 -712.615,E2 -712.615} C_VEL
LIN {X 0,Y 601.421,Z 194.573,A -85,B 0,C 180,E1 -715.308,E2 -715.308} C_VEL
LIN {X 0,Y 601.378,Z 194.57,A -85,B 0,C 180,E1 -717.991,E2 -717.991} C_VEL
LIN {X 0,Y 601.392,Z 194.567,A -85,B 0,C 180,E1 -720,E2 -720} C_VEL
LIN {X 0,Y 601.412,Z 194.567,A -85,B 0,C 180,E1 -722.679,E2 -722.679} C_VEL
LIN {X 0,Y 601.41,Z 194.571,A -85,B 0,C 180,E1 -725.364,E2 -725.364} C_VEL
LIN {X 0,Y 601.369,Z 194.57,A -85,B 0,C 180,E1 -728.062,E2 -728.062} C_VEL
LIN {X 0,Y 601.448,Z 194.57,A -85,B 0,C 180,E1 -731.044,E2 -731.044} C_VEL
LIN {X 0,Y 601.361,Z 194.571,A -85,B 0,C 180,E1 -734.085,E2 -734.085} C_VEL
LIN {X 0,Y 601.396,Z 194.575,A -85,B 0,C 180,E1 -736.987,E2 -736.987} C_VEL
LIN {X 0,Y 601.354,Z 194.572,A -85,B 0,C 180,E1 -739.811,E2 -739.811} C_VEL
LIN {X 0,Y 601.365,Z 194.571,A -85,B 0,C 180,E1 -741.961,E2 -741.961} C_VEL
LIN {X 0,Y 601.358,Z 194.579,A -85,B 0,C 180,E1 -744.881,E2 -744.881} C_VEL
LIN {X 0,Y 601.359,Z 194.572,A -85,B 0,C 180,E1 -747.36,E2 -747.36} C_VEL
LIN {X 0,Y 601.371,Z 194.57,A -85,B 0,C 180,E1 -749.396,E2 -749.396} C_VEL
LIN {X 0,Y 601.368,Z 194.57,A -85,B 0,C 180,E1 -751.729,E2 -751.729} C_VEL
LIN {X 0,Y 601.389,Z 194.572,A -85,B 0,C 180,E1 -754.121,E2 -754.121} C_VEL
LIN {X 0,Y 601.405,Z 194.565,A -85,B 0,C 180,E1 -757.383,E2 -757.383} C_VEL
LIN {X 0,Y 601.409,Z 194.571,A -85,B 0,C 180,E1 -760.577,E2 -760.577} C_VEL
LIN {X 0,Y 601.42,Z 194.568,A -85,B 0,C 180,E1 -762.67,E2 -762.67} C_VEL
LIN {X 0,Y 601.382,Z 194.569,A -85,B 0,C 180,E1 -765.481,E2 -765.481} C_VEL
LIN {X 0,Y 601.408,Z 194.572,A -85,B 0,C 180,E1 -768.409,E2 -768.409} C_VEL
LIN {X 0,Y 601.383,Z 194.569,A -85,B 0,C 180,E1 -770.874,E2 -770.874} C_VEL
LIN {X 0,Y 601.383,Z 194.569,A -85,B 0,C 180,E1 -773.418,E2 -773.418} C_VEL
LIN {X 0,Y 601.425,Z 194.573,A -85,B 0,C 180,E1 -776.066,E2 -776.066} C_VEL
LIN {X 0,Y 601.398,Z 194.567,A -85,B 0,C 180,E1 -779.059,E2 -779.059} C_VEL
LIN {X 0,Y 601.402,Z 194.568,A -85,B 0,C 180,E1 -781.373,E2 -781.373} C_VEL
LIN {X 0,Y 601.414,Z 194.571,A -85,B 0,C 180,E1 -784.133,E2 -784.133} C_VEL
LIN {X 0,Y 601.395,Z 194.571,A -85,B 0,C 180,E1 -786.726,E2 -786.726} C_VEL
LIN {X 0,Y 601.696,Z 199.704,A -85,B 0,C 180,E1 -787.451,E2 -787.451} C_VEL
LIN {X 0,Y 601.598,Z 220.085,A -85,B 0,C 180,E1 -790.198,E2 -790.198} C_VEL
LIN {X 0,Y 601.529,Z 241.356,A -85,B 0,C 180,E1 -793.017,E2 -793.017} C_VEL
LIN {X 0,Y 601.458,Z 262.628,A -85,B 0,C 180,E1 -795.796,E2 -795.796} C_VEL
LIN {X 0,Y 601.425,Z 270.522,A -85,B 0,C 180,E1 -796.818,E2 -796.818} C_VEL
LIN {X 0,Y 601.617,Z 287.242,A -85,B 0,C 180,E1 -797.026,E2 -797.026} C_VEL
LIN {X 0,Y 601.606,Z 378.942,A -85,B 0,C 180,E1 -798.139,E2 -798.139} C_VEL
LIN {X 0,Y 601.569,Z 392.213,A -85,B 0,C 180,E1 -798.438,E2 -798.438} C_VEL
LIN {X 0,Y 601.542,Z 404.639,A -85,B 0,C 180,E1 -798.853,E2 -798.853} C_VEL
LIN {X 0,Y 601.525,Z 416.63,A -85,B 0,C 180,E1 -799.396,E2 -799.396} C_VEL
LIN {X 0,Y 601.486,Z 428.195,A -85,B 0,C 180,E1 -800.076,E2 -800.076} C_VEL
LIN {X 0,Y 601.444,Z 438.591,A -85,B 0,C 180,E1 -800.839,E2 -800.839} C_VEL
LIN {X 0,Y 601.429,Z 447.108,A -85,B 0,C 180,E1 -801.6,E2 -801.6} C_VEL
LIN {X 0,Y 601.418,Z 454.956,A -85,B 0,C 180,E1 -802.445,E2 -802.445} C_VEL
LIN {X 0,Y 601.371,Z 462.222,A -85,B 0,C 180,E1 -803.398,E2 -803.398} C_VEL
LIN {X 0,Y 601.372,Z 467.863,A -85,B 0,C 180,E1 -804.298,E2 -804.298} C_VEL
LIN {X 0,Y 601.336,Z 472.947,A -85,B 0,C 180,E1 -805.307,E2 -805.307} C_VEL
LIN {X 0,Y 601.368,Z 476.893,A -85,B 0,C 180,E1 -806.314,E2 -806.314} C_VEL
LIN {X 0,Y 601.325,Z 479.807,A -85,B 0,C 180,E1 -807.32,E2 -807.32} C_VEL
LIN {X 0,Y 601.343,Z 481.2,A -85,B 0,C 180,E1 -807.99,E2 -807.99} C_VEL
LIN {X 0,Y 601.339,Z 482.783,A -85,B 0,C 180,E1 -809.329,E2 -809.329} C_VEL
LIN {X 0,Y 601.335,Z 483,A -85,B 0,C 180,E1 -809.999,E2 -809.999} C_VEL
LIN {X 0,Y 601.347,Z 482.186,A -85,B 0,C 180,E1 -811.338,E2 -811.338} C_VEL
LIN {X 0,Y 601.343,Z 481.204,A -85,B 0,C 180,E1 -812.008,E2 -812.008} C_VEL
LIN {X 0,Y 601.325,Z 479.813,A -85,B 0,C 180,E1 -812.678,E2 -812.678} C_VEL
LIN {X 0,Y 601.368,Z 476.901,A -85,B 0,C 180,E1 -813.684,E2 -813.684} C_VEL
LIN {X 0,Y 601.336,Z 472.956,A -85,B 0,C 180,E1 -814.691,E2 -814.691} C_VEL
LIN {X 0,Y 601.372,Z 466.887,A -85,B 0,C 180,E1 -815.867,E2 -815.867} C_VEL
LIN {X 0,Y 601.386,Z 460.249,A -85,B 0,C 180,E1 -816.878,E2 -816.878} C_VEL
LIN {X 0,Y 601.4,Z 452.006,A -85,B 0,C 180,E1 -817.89,E2 -817.89} C_VEL
LIN {X 0,Y 601.436,Z 443.559,A -85,B 0,C 180,E1 -818.736,E2 -818.736} C_VEL
LIN {X 0,Y 601.449,Z 433.121,A -85,B 0,C 180,E1 -819.583,E2 -819.583} C_VEL
LIN {X 0,Y 601.473,Z 422.793,A -85,B 0,C 180,E1 -820.262,E2 -820.262} C_VEL
LIN {X 0,Y 601.535,Z 410.624,A -85,B 0,C 180,E1 -820.895,E2 -820.895} C_VEL
LIN {X 0,Y 601.549,Z 398.281,A -85,B 0,C 180,E1 -821.377,E2 -821.377} C_VEL
LIN {X 0,Y 601.571,Z 385.535,A -85,B 0,C 180,E1 -821.731,E2 -821.731} C_VEL
LIN {X 0,Y 601.614,Z 373.255,A -85,B 0,C 180,E1 -821.944,E2 -821.944} C_VEL
LIN {X 0,Y 601.535,Z 271.344,A -85,B 0,C 180,E1 -823.167,E2 -823.167} C_VEL
LIN {X 0,Y 601.431,Z 270.457,A -85,B 0,C 180,E1 -823.191,E2 -823.191} C_VEL
LIN {X 0,Y 601.521,Z 248.022,A -85,B 0,C 180,E1 -826.108,E2 -826.108} C_VEL
LIN {X 0,Y 601.585,Z 225.421,A -85,B 0,C 180,E1 -829.09,E2 -829.09} C_VEL
LIN {X 0,Y 601.677,Z 204.149,A -85,B 0,C 180,E1 -831.946,E2 -831.946} C_VEL
LIN {X 0,Y 601.657,Z 196.172,A -85,B 0,C 180,E1 -833.033,E2 -833.033} C_VEL
LIN {X 0,Y 601.393,Z 194.571,A -85,B 0,C 180,E1 -833.271,E2 -833.271} C_VEL
LIN {X 0,Y 601.414,Z 194.57,A -85,B 0,C 180,E1 -835.867,E2 -835.867} C_VEL
LIN {X 0,Y 601.404,Z 194.568,A -85,B 0,C 180,E1 -838.624,E2 -838.624} C_VEL
LIN {X 0,Y 601.393,Z 194.567,A -85,B 0,C 180,E1 -840.939,E2 -840.939} C_VEL
LIN {X 0,Y 601.424,Z 194.572,A -85,B 0,C 180,E1 -843.934,E2 -843.934} C_VEL
LIN {X 0,Y 601.382,Z 194.57,A -85,B 0,C 180,E1 -846.579,E2 -846.579} C_VEL
LIN {X 0,Y 601.421,Z 194.567,A -85,B 0,C 180,E1 -849.533,E2 -849.533} C_VEL
LIN {X 0,Y 601.407,Z 194.573,A -85,B 0,C 180,E1 -851.76,E2 -851.76} C_VEL
LIN {X 0,Y 601.391,Z 194.568,A -85,B 0,C 180,E1 -854.532,E2 -854.532} C_VEL
LIN {X 0,Y 601.422,Z 194.567,A -85,B 0,C 180,E1 -857.401,E2 -857.401} C_VEL
LIN {X 0,Y 601.403,Z 194.566,A -85,B 0,C 180,E1 -860.46,E2 -860.46} C_VEL
LIN {X 0,Y 601.396,Z 194.566,A -85,B 0,C 180,E1 -862.614,E2 -862.614} C_VEL
LIN {X 0,Y 601.409,Z 194.567,A -85,B 0,C 180,E1 -865.067,E2 -865.067} C_VEL
LIN {X 0,Y 601.428,Z 194.57,A -85,B 0,C 180,E1 -867.484,E2 -867.484} C_VEL
LIN {X 0,Y 601.403,Z 194.572,A -85,B 0,C 180,E1 -869.844,E2 -869.844} C_VEL
LIN {X 0,Y 601.39,Z 194.569,A -85,B 0,C 180,E1 -872.131,E2 -872.131} C_VEL
LIN {X 0,Y 601.379,Z 194.569,A -85,B 0,C 180,E1 -874.38,E2 -874.38} C_VEL
LIN {X 0,Y 601.382,Z 194.568,A -85,B 0,C 180,E1 -876.588,E2 -876.588} C_VEL
LIN {X 0,Y 601.414,Z 194.574,A -85,B 0,C 180,E1 -879.477,E2 -879.477} C_VEL
LIN {X 0,Y 601.388,Z 194.574,A -85,B 0,C 180,E1 -881.607,E2 -881.607} C_VEL
LIN {X 0,Y 601.408,Z 194.569,A -85,B 0,C 180,E1 -883.712,E2 -883.712} C_VEL
LIN {X 0,Y 601.371,Z 194.57,A -85,B 0,C 180,E1 -886.483,E2 -886.483} C_VEL
LIN {X 0,Y 601.408,Z 194.575,A -85,B 0,C 180,E1 -889.224,E2 -889.224} C_VEL
LIN {X 0,Y 601.384,Z 194.569,A -85,B 0,C 180,E1 -891.938,E2 -891.938} C_VEL
LIN {X 0,Y 601.355,Z 194.572,A -85,B 0,C 180,E1 -893.962,E2 -893.962} C_VEL
LIN {X 0,Y 601.393,Z 194.57,A -85,B 0,C 180,E1 -896.65,E2 -896.65} C_VEL
LIN {X 0,Y 601.419,Z 194.57,A -85,B 0,C 180,E1 -899.33,E2 -899.33} C_VEL
LIN {X 0,Y 601.357,Z 194.571,A -85,B 0,C 180,E1 -902.009,E2 -902.009} C_VEL
LIN {X 0,Y 601.384,Z 194.573,A -85,B 0,C 180,E1 -904.692,E2 -904.692} C_VEL
LIN {X 0,Y 601.402,Z 194.569,A -85,B 0,C 180,E1 -907.385,E2 -907.385} C_VEL
LIN {X 0,Y 601.372,Z 194.57,A -85,B 0,C 180,E1 -910.096,E2 -910.096} C_VEL
LIN {X 0,Y 601.356,Z 194.575,A -85,B 0,C 180,E1 -912.402,E2 -912.402} C_VEL
LIN {X 0,Y 600.704,Z 194.662,A -85,B 0,C 180,E1 -912.962,E2 -912.962} C_VEL
LIN {X 0,Y 597.856,Z 195.019,A -85,B 0,C 180,E1 -913.869,E2 -913.869} C_VEL
LIN {X 0,Y 595.439,Z 195.317,A -85,B 0,C 180,E1 -914.6,E2 -914.6} C_VEL
LIN {X 0,Y 594.398,Z 195.443,A -85,B 0,C 180,E1 -915.163,E2 -915.163} C_VEL
LIN {X 0,Y 594.312,Z 195.451,A -85,B 0,C 180,E1 -915.354,E2 -915.354} C_VEL
LIN {X 0,Y 594.338,Z 195.449,A -85,B 0,C 180,E1 -917.195,E2 -917.195} C_VEL
LIN {X 0,Y 594.321,Z 195.45,A -85,B 0,C 180,E1 -919.336,E2 -919.336} C_VEL
LIN {X 0,Y 594.318,Z 195.449,A -85,B 0,C 180,E1 -921.505,E2 -921.505} C_VEL
LIN {X 0,Y 594.34,Z 195.445,A -85,B 0,C 180,E1 -923.706,E2 -923.706} C_VEL
LIN {X 0,Y 594.342,Z 195.454,A -85,B 0,C 180,E1 -926.701,E2 -926.701} C_VEL
LIN {X 0,Y 594.346,Z 195.448,A -85,B 0,C 180,E1 -929,E2 -929} C_VEL
LIN {X 0,Y 594.346,Z 195.445,A -85,B 0,C 180,E1 -931.648,E2 -931.648} C_VEL
LIN {X 0,Y 594.356,Z 195.452,A -85,B 0,C 180,E1 -934.581,E2 -934.581} C_VEL
LIN {X 0,Y 594.343,Z 195.446,A -85,B 0,C 180,E1 -937.089,E2 -937.089} C_VEL
LIN {X 0,Y 594.321,Z 195.449,A -85,B 0,C 180,E1 -939.776,E2 -939.776} C_VEL
LIN {X 0,Y 594.361,Z 195.453,A -85,B 0,C 180,E1 -942.376,E2 -942.376} C_VEL
LIN {X 0,Y 594.307,Z 195.45,A -85,B 0,C 180,E1 -945.197,E2 -945.197} C_VEL
LIN {X 0,Y 594.331,Z 195.448,A -85,B 0,C 180,E1 -947.628,E2 -947.628} C_VEL
LIN {X 0,Y 594.367,Z 195.451,A -85,B 0,C 180,E1 -950.325,E2 -950.325} C_VEL
LIN {X 0,Y 594.354,Z 195.444,A -85,B 0,C 180,E1 -952.916,E2 -952.916} C_VEL
LIN {X 0,Y 594.358,Z 195.449,A -85,B 0,C 180,E1 -955.865,E2 -955.865} C_VEL
LIN {X 0,Y 594.347,Z 195.446,A -85,B 0,C 180,E1 -958.653,E2 -958.653} C_VEL
LIN {X 0,Y 594.356,Z 195.443,A -85,B 0,C 180,E1 -961.047,E2 -961.047} C_VEL
LIN {X 0,Y 594.379,Z 195.451,A -85,B 0,C 180,E1 -963.978,E2 -963.978} C_VEL
LIN {X 0,Y 594.369,Z 195.446,A -85,B 0,C 180,E1 -966.299,E2 -966.299} C_VEL
LIN {X 0,Y 594.377,Z 195.442,A -85,B 0,C 180,E1 -969.227,E2 -969.227} C_VEL
LIN {X 0,Y 594.337,Z 195.452,A -85,B 0,C 180,E1 -972.097,E2 -972.097} C_VEL
LIN {X 0,Y 594.347,Z 195.448,A -85,B 0,C 180,E1 -974.221,E2 -974.221} C_VEL
LIN {X 0,Y 594.366,Z 195.444,A -85,B 0,C 180,E1 -976.323,E2 -976.323} C_VEL
LIN {X 0,Y 594.362,Z 195.443,A -85,B 0,C 180,E1 -978.939,E2 -978.939} C_VEL
LIN {X 0,Y 594.408,Z 195.445,A -85,B 0,C 180,E1 -981.845,E2 -981.845} C_VEL
LIN {X 0,Y 594.371,Z 195.442,A -85,B 0,C 180,E1 -984.574,E2 -984.574} C_VEL
LIN {X 0,Y 594.399,Z 195.615,A -85,B 0,C 180,E1 -986.867,E2 -986.867} C_VEL
LIN {X 0,Y 594.427,Z 209.185,A -85,B 0,C 180,E1 -989.324,E2 -989.324} C_VEL
LIN {X 0,Y 594.361,Z 222.569,A -85,B 0,C 180,E1 -991.716,E2 -991.716} C_VEL
LIN {X 0,Y 594.751,Z 225.724,A -85,B 0,C 180,E1 -991.779,E2 -991.779} C_VEL
LIN {X 0,Y 594.625,Z 329.293,A -85,B 0,C 180,E1 -993.05,E2 -993.05} C_VEL
LIN {X 0,Y 594.59,Z 342.266,A -85,B 0,C 180,E1 -993.347,E2 -993.347} C_VEL
LIN {X 0,Y 594.565,Z 354.772,A -85,B 0,C 180,E1 -993.771,E2 -993.771} C_VEL
LIN {X 0,Y 594.499,Z 366.788,A -85,B 0,C 180,E1 -994.323,E2 -994.323} C_VEL
LIN {X 0,Y 594.425,Z 378.221,A -85,B 0,C 180,E1 -995.003,E2 -995.003} C_VEL
LIN {X 0,Y 594.433,Z 388.516,A -85,B 0,C 180,E1 -995.768,E2 -995.768} C_VEL
LIN {X 0,Y 594.374,Z 398.352,A -85,B 0,C 180,E1 -996.671,E2 -996.671} C_VEL
LIN {X 0,Y 594.322,Z 406.925,A -85,B 0,C 180,E1 -997.645,E2 -997.645} C_VEL
LIN {X 0,Y 594.311,Z 414.248,A -85,B 0,C 180,E1 -998.672,E2 -998.672} C_VEL
LIN {X 0,Y 594.271,Z 419.224,A -85,B 0,C 180,E1 -999.531,E2 -999.531} C_VEL
LIN {X 0,Y 594.288,Z 424.061,A -85,B 0,C 180,E1 -1000.562,E2 -1000.562} C_VEL
LIN {X 0,Y 594.245,Z 427.782,A -85,B 0,C 180,E1 -1001.599,E2 -1001.599} C_VEL
LIN {X 0,Y 594.239,Z 429.703,A -85,B 0,C 180,E1 -1002.291,E2 -1002.291} C_VEL
LIN {X 0,Y 594.243,Z 431.158,A -85,B 0,C 180,E1 -1002.986,E2 -1002.986} C_VEL
LIN {X 0,Y 594.259,Z 432.617,A -85,B 0,C 180,E1 -1004.124,E2 -1004.124} C_VEL
LIN {X 0,Y 594.208,Z 432.997,A -85,B 0,C 180,E1 -1005.082,E2 -1005.082} C_VEL
LIN {X 0,Y 594.222,Z 432.742,A -85,B 0,C 180,E1 -1005.785,E2 -1005.785} C_VEL
LIN {X 0,Y 594.237,Z 431.863,A -85,B 0,C 180,E1 -1006.669,E2 -1006.669} C_VEL
LIN {X 0,Y 594.215,Z 429.414,A -85,B 0,C 180,E1 -1007.909,E2 -1007.909} C_VEL
LIN {X 0,Y 594.243,Z 426.492,A -85,B 0,C 180,E1 -1008.89,E2 -1008.89} C_VEL
LIN {X 0,Y 594.261,Z 421.729,A -85,B 0,C 180,E1 -1010.057,E2 -1010.057} C_VEL
LIN {X 0,Y 594.315,Z 416.024,A -85,B 0,C 180,E1 -1011.128,E2 -1011.128} C_VEL
LIN {X 0,Y 594.313,Z 408.583,A -85,B 0,C 180,E1 -1012.235,E2 -1012.235} C_VEL
LIN {X 0,Y 594.366,Z 400.908,A -85,B 0,C 180,E1 -1013.15,E2 -1013.15} C_VEL
LIN {X 0,Y 594.401,Z 391.435,A -85,B 0,C 180,E1 -1014.073,E2 -1014.073} C_VEL
LIN {X 0,Y 594.457,Z 380.86,A -85,B 0,C 180,E1 -1014.908,E2 -1014.908} C_VEL
LIN {X 0,Y 594.489,Z 370.541,A -85,B 0,C 180,E1 -1015.562,E2 -1015.562} C_VEL
LIN {X 0,Y 594.555,Z 358.46,A -85,B 0,C 180,E1 -1016.164,E2 -1016.164} C_VEL
LIN {X 0,Y 594.562,Z 345.788,A -85,B 0,C 180,E1 -1016.64,E2 -1016.64} C_VEL
LIN {X 0,Y 594.592,Z 332.896,A -85,B 0,C 180,E1 -1016.973,E2 -1016.973} C_VEL
LIN {X 0,Y 594.626,Z 316.876,A -85,B 0,C 180,E1 -1017.209,E2 -1017.209} C_VEL
LIN {X 0,Y 594.619,Z 224.293,A -85,B 0,C 180,E1 -1018.332,E2 -1018.332} C_VEL
LIN {X 0,Y 594.341,Z 222.584,A -85,B 0,C 180,E1 -1018.372,E2 -1018.372} C_VEL
LIN {X 0,Y 594.446,Z 207.073,A -85,B 0,C 180,E1 -1021.146,E2 -1021.146} C_VEL
LIN {X 0,Y 594.407,Z 195.44,A -85,B 0,C 180,E1 -1023.275,E2 -1023.275} C_VEL
LIN {X 0,Y 594.386,Z 195.448,A -85,B 0,C 180,E1 -1026.24,E2 -1026.24} C_VEL
LIN {X 0,Y 594.374,Z 195.445,A -85,B 0,C 180,E1 -1028.803,E2 -1028.803} C_VEL
LIN {X 0,Y 594.374,Z 195.442,A -85,B 0,C 180,E1 -1031.461,E2 -1031.461} C_VEL
LIN {X 0,Y 594.364,Z 195.453,A -85,B 0,C 180,E1 -1034.234,E2 -1034.234} C_VEL
LIN {X 0,Y 594.365,Z 195.443,A -85,B 0,C 180,E1 -1037.144,E2 -1037.144} C_VEL
LIN {X 0,Y 594.367,Z 195.443,A -85,B 0,C 180,E1 -1039.433,E2 -1039.433} C_VEL
LIN {X 0,Y 594.37,Z 195.447,A -85,B 0,C 180,E1 -1042.389,E2 -1042.389} C_VEL
LIN {X 0,Y 594.363,Z 195.444,A -85,B 0,C 180,E1 -1044.67,E2 -1044.67} C_VEL
LIN {X 0,Y 594.36,Z 195.443,A -85,B 0,C 180,E1 -1047.085,E2 -1047.085} C_VEL
LIN {X 0,Y 594.375,Z 195.447,A -85,B 0,C 180,E1 -1049.667,E2 -1049.667} C_VEL
LIN {X 0,Y 594.36,Z 195.444,A -85,B 0,C 180,E1 -1052.539,E2 -1052.539} C_VEL
LIN {X 0,Y 594.352,Z 195.444,A -85,B 0,C 180,E1 -1054.806,E2 -1054.806} C_VEL
LIN {X 0,Y 594.374,Z 195.444,A -85,B 0,C 180,E1 -1057.253,E2 -1057.253} C_VEL
LIN {X 0,Y 594.358,Z 195.449,A -85,B 0,C 180,E1 -1059.946,E2 -1059.946} C_VEL
LIN {X 0,Y 594.354,Z 195.447,A -85,B 0,C 180,E1 -1062.095,E2 -1062.095} C_VEL
LIN {X 0,Y 594.346,Z 195.446,A -85,B 0,C 180,E1 -1064.219,E2 -1064.219} C_VEL
LIN {X 0,Y 594.35,Z 195.447,A -85,B 0,C 180,E1 -1067.017,E2 -1067.017} C_VEL
LIN {X 0,Y 594.368,Z 195.447,A -85,B 0,C 180,E1 -1069.784,E2 -1069.784} C_VEL
LIN {X 0,Y 594.383,Z 195.44,A -85,B 0,C 180,E1 -1072.527,E2 -1072.527} C_VEL
LIN {X 0,Y 594.386,Z 195.448,A -85,B 0,C 180,E1 -1075.253,E2 -1075.253} C_VEL
LIN {X 0,Y 594.35,Z 195.445,A -85,B 0,C 180,E1 -1077.967,E2 -1077.967} C_VEL
LIN {X 0,Y 594.362,Z 195.443,A -85,B 0,C 180,E1 -1080,E2 -1080} C_VEL
LIN {X 0,Y 594.378,Z 195.443,A -85,B 0,C 180,E1 -1082.711,E2 -1082.711} C_VEL
LIN {X 0,Y 594.37,Z 195.446,A -85,B 0,C 180,E1 -1085.428,E2 -1085.428} C_VEL
LIN {X 0,Y 594.364,Z 195.446,A -85,B 0,C 180,E1 -1087.474,E2 -1087.474} C_VEL
LIN {X 0,Y 594.351,Z 195.444,A -85,B 0,C 180,E1 -1090.217,E2 -1090.217} C_VEL
LIN {X 0,Y 594.348,Z 195.445,A -85,B 0,C 180,E1 -1092.289,E2 -1092.289} C_VEL
LIN {X 0,Y 594.337,Z 195.453,A -85,B 0,C 180,E1 -1095.079,E2 -1095.079} C_VEL
LIN {X 0,Y 594.351,Z 195.449,A -85,B 0,C 180,E1 -1097.195,E2 -1097.195} C_VEL
LIN {X 0,Y 594.333,Z 195.447,A -85,B 0,C 180,E1 -1100.055,E2 -1100.055} C_VEL
LIN {X 0,Y 594.321,Z 195.454,A -85,B 0,C 180,E1 -1102.969,E2 -1102.969} C_VEL
LIN {X 0,Y 594.32,Z 195.451,A -85,B 0,C 180,E1 -1105.196,E2 -1105.196} C_VEL
LIN {X 0,Y 594.311,Z 195.449,A -85,B 0,C 180,E1 -1107.52,E2 -1107.52} C_VEL
LIN {X 0,Y 594.329,Z 195.447,A -85,B 0,C 180,E1 -1109.779,E2 -1109.779} C_VEL
LIN {X 0,Y 594.345,Z 195.449,A -85,B 0,C 180,E1 -1112.149,E2 -1112.149} C_VEL
LIN {X 0,Y 594.35,Z 195.453,A -85,B 0,C 180,E1 -1114.582,E2 -1114.582} C_VEL
LIN {X 0,Y 594.361,Z 195.443,A -85,B 0,C 180,E1 -1117.61,E2 -1117.61} C_VEL
LIN {X 0,Y 594.363,Z 195.449,A -85,B 0,C 180,E1 -1120.568,E2 -1120.568} C_VEL
LIN {X 0,Y 594.339,Z 195.446,A -85,B 0,C 180,E1 -1123.302,E2 -1123.302} C_VEL
LIN {X 0,Y 594.345,Z 195.454,A -85,B 0,C 180,E1 -1126.163,E2 -1126.163} C_VEL
LIN {X 0,Y 594.352,Z 195.444,A -85,B 0,C 180,E1 -1129.181,E2 -1129.181} C_VEL
LIN {X 0,Y 594.367,Z 195.452,A -85,B 0,C 180,E1 -1132.061,E2 -1132.061} C_VEL
LIN {X 0,Y 594.341,Z 195.447,A -85,B 0,C 180,E1 -1134.678,E2 -1134.678} C_VEL
LIN {X 0,Y 594.366,Z 195.443,A -85,B 0,C 180,E1 -1137.091,E2 -1137.091} C_VEL
LIN {X 0,Y 594.38,Z 195.447,A -85,B 0,C 180,E1 -1139.673,E2 -1139.673} C_VEL
LIN {X 0,Y 594.372,Z 195.444,A -85,B 0,C 180,E1 -1142.54,E2 -1142.54} C_VEL
LIN {X 0,Y 594.397,Z 195.446,A -85,B 0,C 180,E1 -1145.565,E2 -1145.565} C_VEL
LIN {X 0,Y 594.362,Z 195.489,A -85,B 0,C 180,E1 -1146.573,E2 -1146.573} C_VEL
LIN {X 0,Y 594.786,Z 199.667,A -85,B 0,C 180,E1 -1147.169,E2 -1147.169} C_VEL
LIN {X 0,Y 594.669,Z 220.085,A -85,B 0,C 180,E1 -1149.957,E2 -1149.957} C_VEL
LIN {X 0,Y 594.564,Z 240.027,A -85,B 0,C 180,E1 -1152.635,E2 -1152.635} C_VEL
LIN {X 0,Y 594.472,Z 261.299,A -85,B 0,C 180,E1 -1155.45,E2 -1155.45} C_VEL
LIN {X 0,Y 594.434,Z 270.439,A -85,B 0,C 180,E1 -1156.649,E2 -1156.649} C_VEL
LIN {X 0,Y 594.732,Z 276.511,A -85,B 0,C 180,E1 -1156.743,E2 -1156.743} C_VEL
LIN {X 0,Y 594.657,Z 378.942,A -85,B 0,C 180,E1 -1157.999,E2 -1157.999} C_VEL
LIN {X 0,Y 594.631,Z 392.214,A -85,B 0,C 180,E1 -1158.301,E2 -1158.301} C_VEL
LIN {X 0,Y 594.597,Z 404.432,A -85,B 0,C 180,E1 -1158.713,E2 -1158.713} C_VEL
LIN {X 0,Y 594.528,Z 416.628,A -85,B 0,C 180,E1 -1159.27,E2 -1159.27} C_VEL
LIN {X 0,Y 594.48,Z 428.197,A -85,B 0,C 180,E1 -1159.957,E2 -1159.957} C_VEL
LIN {X 0,Y 594.414,Z 438.593,A -85,B 0,C 180,E1 -1160.729,E2 -1160.729} C_VEL
LIN {X 0,Y 594.383,Z 447.108,A -85,B 0,C 180,E1 -1161.5,E2 -1161.5} C_VEL
LIN {X 0,Y 594.347,Z 454.956,A -85,B 0,C 180,E1 -1162.355,E2 -1162.355} C_VEL
LIN {X 0,Y 594.283,Z 462.811,A -85,B 0,C 180,E1 -1163.408,E2 -1163.408} C_VEL
LIN {X 0,Y 594.289,Z 469.677,A -85,B 0,C 180,E1 -1164.571,E2 -1164.571} C_VEL
LIN {X 0,Y 594.27,Z 474.368,A -85,B 0,C 180,E1 -1165.591,E2 -1165.591} C_VEL
LIN {X 0,Y 594.267,Z 477.954,A -85,B 0,C 180,E1 -1166.609,E2 -1166.609} C_VEL
LIN {X 0,Y 594.226,Z 479.806,A -85,B 0,C 180,E1 -1167.287,E2 -1167.287} C_VEL
LIN {X 0,Y 594.242,Z 481.199,A -85,B 0,C 180,E1 -1167.966,E2 -1167.966} C_VEL
LIN {X 0,Y 594.239,Z 482.783,A -85,B 0,C 180,E1 -1169.321,E2 -1169.321} C_VEL
LIN {X 0,Y 594.236,Z 483,A -85,B 0,C 180,E1 -1169.999,E2 -1169.999} C_VEL
LIN {X 0,Y 594.247,Z 482.186,A -85,B 0,C 180,E1 -1171.354,E2 -1171.354} C_VEL
LIN {X 0,Y 594.242,Z 481.204,A -85,B 0,C 180,E1 -1172.032,E2 -1172.032} C_VEL
LIN {X 0,Y 594.225,Z 479.813,A -85,B 0,C 180,E1 -1172.71,E2 -1172.71} C_VEL
LIN {X 0,Y 594.289,Z 476.901,A -85,B 0,C 180,E1 -1173.728,E2 -1173.728} C_VEL
LIN {X 0,Y 594.241,Z 472.956,A -85,B 0,C 180,E1 -1174.747,E2 -1174.747} C_VEL
LIN {X 0,Y 594.304,Z 466.888,A -85,B 0,C 180,E1 -1175.938,E2 -1175.938} C_VEL
LIN {X 0,Y 594.31,Z 460.25,A -85,B 0,C 180,E1 -1176.96,E2 -1176.96} C_VEL
LIN {X 0,Y 594.358,Z 452.007,A -85,B 0,C 180,E1 -1177.984,E2 -1177.984} C_VEL
LIN {X 0,Y 594.381,Z 443.56,A -85,B 0,C 180,E1 -1178.84,E2 -1178.84} C_VEL
LIN {X 0,Y 594.433,Z 433.123,A -85,B 0,C 180,E1 -1179.697,E2 -1179.697} C_VEL
LIN {X 0,Y 594.485,Z 422.794,A -85,B 0,C 180,E1 -1180.384,E2 -1180.384} C_VEL
LIN {X 0,Y 594.558,Z 411.726,A -85,B 0,C 180,E1 -1180.973,E2 -1180.973} C_VEL
LIN {X 0,Y 594.574,Z 399.766,A -85,B 0,C 180,E1 -1181.462,E2 -1181.462} C_VEL
LIN {X 0,Y 594.635,Z 386.448,A -85,B 0,C 180,E1 -1181.848,E2 -1181.848} C_VEL
LIN {X 0,Y 594.692,Z 373.255,A -85,B 0,C 180,E1 -1182.085,E2 -1182.085} C_VEL
LIN {X 0,Y 594.626,Z 272.014,A -85,B 0,C 180,E1 -1183.314,E2 -1183.314} C_VEL
LIN {X 0,Y 594.433,Z 270.457,A -85,B 0,C 180,E1 -1183.349,E2 -1183.349} C_VEL
LIN {X 0,Y 594.537,Z 248.022,A -85,B 0,C 180,E1 -1186.302,E2 -1186.302} C_VEL
LIN {X 0,Y 594.619,Z 227.111,A -85,B 0,C 180,E1 -1189.095,E2 -1189.095} C_VEL
LIN {X 0,Y 594.76,Z 206.808,A -85,B 0,C 180,E1 -1191.849,E2 -1191.849} C_VEL
LIN {X 0,Y 594.739,Z 197.502,A -85,B 0,C 180,E1 -1193.132,E2 -1193.132} C_VEL
LIN {X 0,Y 594.345,Z 195.451,A -85,B 0,C 180,E1 -1193.471,E2 -1193.471} C_VEL
LIN {X 0,Y 594.384,Z 195.449,A -85,B 0,C 180,E1 -1196.022,E2 -1196.022} C_VEL
LIN {X 0,Y 594.361,Z 195.443,A -85,B 0,C 180,E1 -1198.995,E2 -1198.995} C_VEL
LIN {X 0,Y 594.361,Z 195.446,A -85,B 0,C 180,E1 -1201.64,E2 -1201.64} C_VEL
LIN {X 0,Y 594.368,Z 195.444,A -85,B 0,C 180,E1 -1204.576,E2 -1204.576} C_VEL
LIN {X 0,Y 594.359,Z 195.443,A -85,B 0,C 180,E1 -1207.083,E2 -1207.083} C_VEL
LIN {X 0,Y 594.355,Z 195.451,A -85,B 0,C 180,E1 -1209.771,E2 -1209.771} C_VEL
LIN {X 0,Y 594.34,Z 195.448,A -85,B 0,C 180,E1 -1212.372,E2 -1212.372} C_VEL
LIN {X 0,Y 594.33,Z 195.448,A -85,B 0,C 180,E1 -1215.188,E2 -1215.188} C_VEL
LIN {X 0,Y 594.367,Z 195.45,A -85,B 0,C 180,E1 -1217.624,E2 -1217.624} C_VEL
LIN {X 0,Y 594.366,Z 195.444,A -85,B 0,C 180,E1 -1220.319,E2 -1220.319} C_VEL
LIN {X 0,Y 594.348,Z 195.445,A -85,B 0,C 180,E1 -1222.91,E2 -1222.91} C_VEL
LIN {X 0,Y 594.351,Z 195.451,A -85,B 0,C 180,E1 -1225.856,E2 -1225.856} C_VEL
LIN {X 0,Y 594.348,Z 195.444,A -85,B 0,C 180,E1 -1228.648,E2 -1228.648} C_VEL
LIN {X 0,Y 594.38,Z 195.443,A -85,B 0,C 180,E1 -1231.031,E2 -1231.031} C_VEL
LIN {X 0,Y 594.332,Z 195.449,A -85,B 0,C 180,E1 -1234.054,E2 -1234.054} C_VEL
LIN {X 0,Y 594.368,Z 195.445,A -85,B 0,C 180,E1 -1237.033,E2 -1237.033} C_VEL
LIN {X 0,Y 594.34,Z 195.448,A -85,B 0,C 180,E1 -1239.945,E2 -1239.945} C_VEL
LIN {X 0,Y 594.336,Z 195.447,A -85,B 0,C 180,E1 -1242.094,E2 -1242.094} C_VEL
LIN {X 0,Y 594.326,Z 195.447,A -85,B 0,C 180,E1 -1244.218,E2 -1244.218} C_VEL
LIN {X 0,Y 594.356,Z 195.449,A -85,B 0,C 180,E1 -1247.017,E2 -1247.017} C_VEL
LIN {X 0,Y 594.376,Z 195.449,A -85,B 0,C 180,E1 -1249.094,E2 -1249.094} C_VEL
LIN {X 0,Y 594.363,Z 195.444,A -85,B 0,C 180,E1 -1251.842,E2 -1251.842} C_VEL
LIN {X 0,Y 594.314,Z 195.449,A -85,B 0,C 180,E1 -1253.89,E2 -1253.89} C_VEL
LIN {X 0,Y 594.302,Z 195.451,A -85,B 0,C 180,E1 -1255.931,E2 -1255.931} C_VEL
LIN {X 0,Y 594.331,Z 195.447,A -85,B 0,C 180,E1 -1257.967,E2 -1257.967} C_VEL
LIN {X 0,Y 594.381,Z 195.444,A -85,B 0,C 180,E1 -1260.677,E2 -1260.677} C_VEL
LIN {X 0,Y 594.346,Z 195.449,A -85,B 0,C 180,E1 -1263.389,E2 -1263.389} C_VEL
LIN {X 0,Y 594.303,Z 195.45,A -85,B 0,C 180,E1 -1266.109,E2 -1266.109} C_VEL
LIN {X 0,Y 594.353,Z 195.444,A -85,B 0,C 180,E1 -1268.157,E2 -1268.157} C_VEL
LIN {X 0,Y 594.403,Z 195.444,A -85,B 0,C 180,E1 -1271.113,E2 -1271.113} C_VEL
LIN {X 0,Y 594.332,Z 195.45,A -85,B 0,C 180,E1 -1274.378,E2 -1274.378} C_VEL
LIN {X 0,Y 594.312,Z 195.451,A -85,B 0,C 180,E1 -1275.354,E2 -1275.354} C_VEL
LIN {X 0,Y 593.639,Z 195.535,A -85,B 0,C 180,E1 -1275.92,E2 -1275.92} C_VEL
LIN {X 0,Y 590.781,Z 195.899,A -85,B 0,C 180,E1 -1276.838,E2 -1276.838} C_VEL
LIN {X 0,Y 588.377,Z 196.193,A -85,B 0,C 180,E1 -1277.577,E2 -1277.577} C_VEL
LIN {X 0,Y 587.357,Z 196.317,A -85,B 0,C 180,E1 -1278.147,E2 -1278.147} C_VEL
LIN {X 0,Y 587.28,Z 196.327,A -85,B 0,C 180,E1 -1278.34,E2 -1278.34} C_VEL
LIN {X 0,Y 587.301,Z 196.327,A -85,B 0,C 180,E1 -1281.047,E2 -1281.047} C_VEL
LIN {X 0,Y 587.313,Z 196.323,A -85,B 0,C 180,E1 -1283.259,E2 -1283.259} C_VEL
LIN {X 0,Y 587.31,Z 196.326,A -85,B 0,C 180,E1 -1286.28,E2 -1286.28} C_VEL
LIN {X 0,Y 587.31,Z 196.323,A -85,B 0,C 180,E1 -1289.138,E2 -1289.138} C_VEL
LIN {X 0,Y 587.314,Z 196.322,A -85,B 0,C 180,E1 -1291.841,E2 -1291.841} C_VEL
LIN {X 0,Y 587.311,Z 196.329,A -85,B 0,C 180,E1 -1294.352,E2 -1294.352} C_VEL
LIN {X 0,Y 587.31,Z 196.326,A -85,B 0,C 180,E1 -1296.749,E2 -1296.749} C_VEL
LIN {X 0,Y 587.292,Z 196.323,A -85,B 0,C 180,E1 -1299.363,E2 -1299.363} C_VEL
LIN {X 0,Y 587.328,Z 196.325,A -85,B 0,C 180,E1 -1302.115,E2 -1302.115} C_VEL
LIN {X 0,Y 587.263,Z 196.328,A -85,B 0,C 180,E1 -1305.09,E2 -1305.09} C_VEL
LIN {X 0,Y 587.32,Z 196.325,A -85,B 0,C 180,E1 -1307.931,E2 -1307.931} C_VEL
LIN {X 0,Y 587.298,Z 196.323,A -85,B 0,C 180,E1 -1311.062,E2 -1311.062} C_VEL
LIN {X 0,Y 587.325,Z 196.32,A -85,B 0,C 180,E1 -1313.295,E2 -1313.295} C_VEL
LIN {X 0,Y 587.336,Z 196.323,A -85,B 0,C 180,E1 -1315.783,E2 -1315.783} C_VEL
LIN {X 0,Y 587.317,Z 196.328,A -85,B 0,C 180,E1 -1318.234,E2 -1318.234} C_VEL
LIN {X 0,Y 587.327,Z 196.319,A -85,B 0,C 180,E1 -1320.87,E2 -1320.87} C_VEL
LIN {X 0,Y 587.346,Z 196.324,A -85,B 0,C 180,E1 -1323.821,E2 -1323.821} C_VEL
LIN {X 0,Y 587.32,Z 196.33,A -85,B 0,C 180,E1 -1325.996,E2 -1325.996} C_VEL
LIN {X 0,Y 587.304,Z 196.327,A -85,B 0,C 180,E1 -1328.228,E2 -1328.228} C_VEL
LIN {X 0,Y 587.323,Z 196.32,A -85,B 0,C 180,E1 -1331.153,E2 -1331.153} C_VEL
LIN {X 0,Y 587.3,Z 196.329,A -85,B 0,C 180,E1 -1334.027,E2 -1334.027} C_VEL
LIN {X 0,Y 587.346,Z 196.321,A -85,B 0,C 180,E1 -1336.156,E2 -1336.156} C_VEL
LIN {X 0,Y 587.332,Z 196.319,A -85,B 0,C 180,E1 -1338.964,E2 -1338.964} C_VEL
LIN {X 0,Y 587.359,Z 196.325,A -85,B 0,C 180,E1 -1341.747,E2 -1341.747} C_VEL
LIN {X 0,Y 587.341,Z 196.318,A -85,B 0,C 180,E1 -1344.509,E2 -1344.509} C_VEL
LIN {X 0,Y 587.324,Z 196.406,A -85,B 0,C 180,E1 -1346.786,E2 -1346.786} C_VEL
LIN {X 0,Y 587.395,Z 208.32,A -85,B 0,C 180,E1 -1348.973,E2 -1348.973} C_VEL
LIN {X 0,Y 587.329,Z 222.634,A -85,B 0,C 180,E1 -1351.565,E2 -1351.565} C_VEL
LIN {X 0,Y 587.852,Z 226.386,A -85,B 0,C 180,E1 -1351.628,E2 -1351.628} C_VEL
LIN {X 0,Y 587.693,Z 329.716,A -85,B 0,C 180,E1 -1352.914,E2 -1352.914} C_VEL
LIN {X 0,Y 587.647,Z 342.551,A -85,B 0,C 180,E1 -1353.215,E2 -1353.215} C_VEL
LIN {X 0,Y 587.593,Z 354.996,A -85,B 0,C 180,E1 -1353.644,E2 -1353.644} C_VEL
LIN {X 0,Y 587.521,Z 366.941,A -85,B 0,C 180,E1 -1354.203,E2 -1354.203} C_VEL
LIN {X 0,Y 587.401,Z 378.359,A -85,B 0,C 180,E1 -1354.891,E2 -1354.891} C_VEL
LIN {X 0,Y 587.399,Z 388.629,A -85,B 0,C 180,E1 -1355.665,E2 -1355.665} C_VEL
LIN {X 0,Y 587.335,Z 398.457,A -85,B 0,C 180,E1 -1356.581,E2 -1356.581} C_VEL
LIN {X 0,Y 587.261,Z 406.997,A -85,B 0,C 180,E1 -1357.565,E2 -1357.565} C_VEL
LIN {X 0,Y 587.247,Z 414.304,A -85,B 0,C 180,E1 -1358.604,E2 -1358.604} C_VEL
LIN {X 0,Y 587.2,Z 420.182,A -85,B 0,C 180,E1 -1359.646,E2 -1359.646} C_VEL
LIN {X 0,Y 587.188,Z 424.817,A -85,B 0,C 180,E1 -1360.692,E2 -1360.692} C_VEL
LIN {X 0,Y 587.162,Z 428.347,A -85,B 0,C 180,E1 -1361.741,E2 -1361.741} C_VEL
LIN {X 0,Y 587.159,Z 430.118,A -85,B 0,C 180,E1 -1362.442,E2 -1362.442} C_VEL
LIN {X 0,Y 587.144,Z 431.457,A -85,B 0,C 180,E1 -1363.146,E2 -1363.146} C_VEL
LIN {X 0,Y 587.157,Z 432.663,A -85,B 0,C 180,E1 -1364.18,E2 -1364.18} C_VEL
LIN {X 0,Y 587.122,Z 432.956,A -85,B 0,C 180,E1 -1365.268,E2 -1365.268} C_VEL
LIN {X 0,Y 587.136,Z 432.614,A -85,B 0,C 180,E1 -1365.98,E2 -1365.98} C_VEL
LIN {X 0,Y 587.141,Z 431.773,A -85,B 0,C 180,E1 -1366.747,E2 -1366.747} C_VEL
LIN {X 0,Y 587.133,Z 430.611,A -85,B 0,C 180,E1 -1367.412,E2 -1367.412} C_VEL
LIN {X 0,Y 587.162,Z 427.906,A -85,B 0,C 180,E1 -1368.493,E2 -1368.493} C_VEL
LIN {X 0,Y 587.167,Z 424.069,A -85,B 0,C 180,E1 -1369.581,E2 -1369.581} C_VEL
LIN {X 0,Y 587.183,Z 419.062,A -85,B 0,C 180,E1 -1370.657,E2 -1370.657} C_VEL
LIN {X 0,Y 587.228,Z 412.418,A -85,B 0,C 180,E1 -1371.777,E2 -1371.777} C_VEL
LIN {X 0,Y 587.26,Z 405.698,A -85,B 0,C 180,E1 -1372.69,E2 -1372.69} C_VEL
LIN {X 0,Y 587.333,Z 397.28,A -85,B 0,C 180,E1 -1373.631,E2 -1373.631} C_VEL
LIN {X 0,Y 587.398,Z 387.58,A -85,B 0,C 180,E1 -1374.511,E2 -1374.511} C_VEL
LIN {X 0,Y 587.44,Z 376.545,A -85,B 0,C 180,E1 -1375.321,E2 -1375.321} C_VEL
LIN {X 0,Y 587.562,Z 365.145,A -85,B 0,C 180,E1 -1375.98,E2 -1375.98} C_VEL
LIN {X 0,Y 587.593,Z 352.277,A -85,B 0,C 180,E1 -1376.552,E2 -1376.552} C_VEL
LIN {X 0,Y 587.634,Z 339.692,A -85,B 0,C 180,E1 -1376.958,E2 -1376.958} C_VEL
LIN {X 0,Y 587.667,Z 327.102,A -85,B 0,C 180,E1 -1377.22,E2 -1377.22} C_VEL
LIN {X 0,Y 587.79,Z 225.581,A -85,B 0,C 180,E1 -1378.473,E2 -1378.473} C_VEL
LIN {X 0,Y 587.311,Z 222.587,A -85,B 0,C 180,E1 -1378.534,E2 -1378.534} C_VEL
LIN {X 0,Y 587.409,Z 208.081,A -85,B 0,C 180,E1 -1381.16,E2 -1381.16} C_VEL
LIN {X 0,Y 587.361,Z 196.319,A -85,B 0,C 180,E1 -1383.331,E2 -1383.331} C_VEL
LIN {X 0,Y 587.347,Z 196.32,A -85,B 0,C 180,E1 -1385.894,E2 -1385.894} C_VEL
LIN {X 0,Y 587.321,Z 196.329,A -85,B 0,C 180,E1 -1388.477,E2 -1388.477} C_VEL
LIN {X 0,Y 587.348,Z 196.317,A -85,B 0,C 180,E1 -1391.153,E2 -1391.153} C_VEL
LIN {X 0,Y 587.317,Z 196.329,A -85,B 0,C 180,E1 -1394.113,E2 -1394.113} C_VEL
LIN {X 0,Y 587.317,Z 196.321,A -85,B 0,C 180,E1 -1396.994,E2 -1396.994} C_VEL
LIN {X 0,Y 587.31,Z 196.329,A -85,B 0,C 180,E1 -1399.978,E2 -1399.978} C_VEL
LIN {X 0,Y 587.325,Z 196.324,A -85,B 0,C 180,E1 -1402.391,E2 -1402.391} C_VEL
LIN {X 0,Y 587.329,Z 196.319,A -85,B 0,C 180,E1 -1404.945,E2 -1404.945} C_VEL
LIN {X 0,Y 587.324,Z 196.322,A -85,B 0,C 180,E1 -1407.42,E2 -1407.42} C_VEL
LIN {X 0,Y 587.322,Z 196.328,A -85,B 0,C 180,E1 -1409.829,E2 -1409.829} C_VEL
LIN {X 0,Y 587.323,Z 196.323,A -85,B 0,C 180,E1 -1412.305,E2 -1412.305} C_VEL
LIN {X 0,Y 587.311,Z 196.322,A -85,B 0,C 180,E1 -1414.483,E2 -1414.483} C_VEL
LIN {X 0,Y 587.342,Z 196.323,A -85,B 0,C 180,E1 -1417.487,E2 -1417.487} C_VEL
LIN {X 0,Y 587.321,Z 196.321,A -85,B 0,C 180,E1 -1420.424,E2 -1420.424} C_VEL
LIN {X 0,Y 587.349,Z 196.321,A -85,B 0,C 180,E1 -1423.311,E2 -1423.311} C_VEL
LIN {X 0,Y 587.332,Z 196.32,A -85,B 0,C 180,E1 -1426.154,E2 -1426.154} C_VEL
LIN {X 0,Y 587.326,Z 196.321,A -85,B 0,C 180,E1 -1428.962,E2 -1428.962} C_VEL
LIN {X 0,Y 587.339,Z 196.322,A -85,B 0,C 180,E1 -1431.745,E2 -1431.745} C_VEL
LIN {X 0,Y 587.293,Z 196.327,A -85,B 0,C 180,E1 -1433.817,E2 -1433.817} C_VEL
LIN {X 0,Y 587.278,Z 196.327,A -85,B 0,C 180,E1 -1435.883,E2 -1435.883} C_VEL
LIN {X 0,Y 587.322,Z 196.321,A -85,B 0,C 180,E1 -1437.943,E2 -1437.943} C_VEL
LIN {X 0,Y 587.333,Z 196.319,A -85,B 0,C 180,E1 -1440,E2 -1440} C_VEL
LIN {X 0,Y 587.345,Z 196.32,A -85,B 0,C 180,E1 -1442.744,E2 -1442.744} C_VEL
LIN {X 0,Y 587.331,Z 196.322,A -85,B 0,C 180,E1 -1445.493,E2 -1445.493} C_VEL
LIN {X 0,Y 587.293,Z 196.323,A -85,B 0,C 180,E1 -1448.257,E2 -1448.257} C_VEL
LIN {X 0,Y 587.375,Z 196.32,A -85,B 0,C 180,E1 -1451.167,E2 -1451.167} C_VEL
LIN {X 0,Y 587.301,Z 196.326,A -85,B 0,C 180,E1 -1454.555,E2 -1454.555} C_VEL
LIN {X 0,Y 587.309,Z 196.324,A -85,B 0,C 180,E1 -1457.407,E2 -1457.407} C_VEL
LIN {X 0,Y 587.273,Z 196.326,A -85,B 0,C 180,E1 -1459.578,E2 -1459.578} C_VEL
LIN {X 0,Y 587.281,Z 196.325,A -85,B 0,C 180,E1 -1461.776,E2 -1461.776} C_VEL
LIN {X 0,Y 587.275,Z 196.335,A -85,B 0,C 180,E1 -1464.762,E2 -1464.762} C_VEL
LIN {X 0,Y 587.284,Z 196.328,A -85,B 0,C 180,E1 -1467.049,E2 -1467.049} C_VEL
LIN {X 0,Y 587.31,Z 196.322,A -85,B 0,C 180,E1 -1469.382,E2 -1469.382} C_VEL
LIN {X 0,Y 587.315,Z 196.321,A -85,B 0,C 180,E1 -1471.837,E2 -1471.837} C_VEL
LIN {X 0,Y 587.314,Z 196.329,A -85,B 0,C 180,E1 -1474.348,E2 -1474.348} C_VEL
LIN {X 0,Y 587.316,Z 196.321,A -85,B 0,C 180,E1 -1477.61,E2 -1477.61} C_VEL
LIN {X 0,Y 587.296,Z 196.332,A -85,B 0,C 180,E1 -1480.256,E2 -1480.256} C_VEL
LIN {X 0,Y 587.303,Z 196.323,A -85,B 0,C 180,E1 -1483.008,E2 -1483.008} C_VEL
LIN {X 0,Y 587.297,Z 196.33,A -85,B 0,C 180,E1 -1486.05,E2 -1486.05} C_VEL
LIN {X 0,Y 587.318,Z 196.321,A -85,B 0,C 180,E1 -1488.927,E2 -1488.927} C_VEL
LIN {X 0,Y 587.305,Z 196.324,A -85,B 0,C 180,E1 -1491.521,E2 -1491.521} C_VEL
LIN {X 0,Y 587.293,Z 196.334,A -85,B 0,C 180,E1 -1494.102,E2 -1494.102} C_VEL
LIN {X 0,Y 587.329,Z 196.32,A -85,B 0,C 180,E1 -1496.89,E2 -1496.89} C_VEL
LIN {X 0,Y 587.326,Z 196.328,A -85,B 0,C 180,E1 -1499.831,E2 -1499.831} C_VEL
LIN {X 0,Y 587.301,Z 196.327,A -85,B 0,C 180,E1 -1502.317,E2 -1502.317} C_VEL
LIN {X 0,Y 587.346,Z 196.32,A -85,B 0,C 180,E1 -1505.242,E2 -1505.242} C_VEL
LIN {X 0,Y 587.343,Z 196.384,A -85,B 0,C 180,E1 -1506.416,E2 -1506.416} C_VEL
LIN {X 0,Y 587.882,Z 200.503,A -85,B 0,C 180,E1 -1507.002,E2 -1507.002} C_VEL
LIN {X 0,Y 587.761,Z 220.085,A -85,B 0,C 180,E1 -1509.711,E2 -1509.711} C_VEL
LIN {X 0,Y 587.575,Z 241.356,A -85,B 0,C 180,E1 -1512.601,E2 -1512.601} C_VEL
LIN {X 0,Y 587.475,Z 261.299,A -85,B 0,C 180,E1 -1515.273,E2 -1515.273} C_VEL
LIN {X 0,Y 587.402,Z 270.439,A -85,B 0,C 180,E1 -1516.486,E2 -1516.486} C_VEL
LIN {X 0,Y 587.84,Z 274.722,A -85,B 0,C 180,E1 -1516.562,E2 -1516.562} C_VEL
LIN {X 0,Y 587.72,Z 378.942,A -85,B 0,C 180,E1 -1517.855,E2 -1517.855} C_VEL
LIN {X 0,Y 587.681,Z 392.215,A -85,B 0,C 180,E1 -1518.16,E2 -1518.16} C_VEL
LIN {X 0,Y 587.629,Z 404.602,A -85,B 0,C 180,E1 -1518.584,E2 -1518.584} C_VEL
LIN {X 0,Y 587.53,Z 416.626,A -85,B 0,C 180,E1 -1519.14,E2 -1519.14} C_VEL
LIN {X 0,Y 587.468,Z 428.199,A -85,B 0,C 180,E1 -1519.836,E2 -1519.836} C_VEL
LIN {X 0,Y 587.394,Z 438.594,A -85,B 0,C 180,E1 -1520.617,E2 -1520.617} C_VEL
LIN {X 0,Y 587.322,Z 447.108,A -85,B 0,C 180,E1 -1521.397,E2 -1521.397} C_VEL
LIN {X 0,Y 587.274,Z 454.956,A -85,B 0,C 180,E1 -1522.262,E2 -1522.262} C_VEL
LIN {X 0,Y 587.231,Z 461.465,A -85,B 0,C 180,E1 -1523.126,E2 -1523.126} C_VEL
LIN {X 0,Y 587.236,Z 467.863,A -85,B 0,C 180,E1 -1524.161,E2 -1524.161} C_VEL
LIN {X 0,Y 587.147,Z 472.947,A -85,B 0,C 180,E1 -1525.193,E2 -1525.193} C_VEL
LIN {X 0,Y 587.213,Z 476.893,A -85,B 0,C 180,E1 -1526.225,E2 -1526.225} C_VEL
LIN {X 0,Y 587.132,Z 479.806,A -85,B 0,C 180,E1 -1527.255,E2 -1527.255} C_VEL
LIN {X 0,Y 587.141,Z 481.198,A -85,B 0,C 180,E1 -1527.941,E2 -1527.941} C_VEL
LIN {X 0,Y 587.14,Z 482.784,A -85,B 0,C 180,E1 -1529.313,E2 -1529.313} C_VEL
LIN {X 0,Y 587.137,Z 483,A -85,B 0,C 180,E1 -1529.999,E2 -1529.999} C_VEL
LIN {X 0,Y 587.147,Z 482.187,A -85,B 0,C 180,E1 -1531.37,E2 -1531.37} C_VEL
LIN {X 0,Y 587.141,Z 481.203,A -85,B 0,C 180,E1 -1532.057,E2 -1532.057} C_VEL
LIN {X 0,Y 587.132,Z 479.813,A -85,B 0,C 180,E1 -1532.743,E2 -1532.743} C_VEL
LIN {X 0,Y 587.213,Z 476.901,A -85,B 0,C 180,E1 -1533.773,E2 -1533.773} C_VEL
LIN {X 0,Y 587.147,Z 472.956,A -85,B 0,C 180,E1 -1534.805,E2 -1534.805} C_VEL
LIN {X 0,Y 587.236,Z 467.876,A -85,B 0,C 180,E1 -1535.837,E2 -1535.837} C_VEL
LIN {X 0,Y 587.231,Z 461.482,A -85,B 0,C 180,E1 -1536.872,E2 -1536.872} C_VEL
LIN {X 0,Y 587.286,Z 453.495,A -85,B 0,C 180,E1 -1537.908,E2 -1537.908} C_VEL
LIN {X 0,Y 587.335,Z 445.357,A -85,B 0,C 180,E1 -1538.774,E2 -1538.774} C_VEL
LIN {X 0,Y 587.391,Z 435.428,A -85,B 0,C 180,E1 -1539.641,E2 -1539.641} C_VEL
LIN {X 0,Y 587.482,Z 424.209,A -85,B 0,C 180,E1 -1540.422,E2 -1540.422} C_VEL
LIN {X 0,Y 587.58,Z 412.558,A -85,B 0,C 180,E1 -1541.064,E2 -1541.064} C_VEL
LIN {X 0,Y 587.61,Z 400.018,A -85,B 0,C 180,E1 -1541.592,E2 -1541.592} C_VEL
LIN {X 0,Y 587.689,Z 387.361,A -85,B 0,C 180,E1 -1541.968,E2 -1541.968} C_VEL
LIN {X 0,Y 587.75,Z 374.763,A -85,B 0,C 180,E1 -1542.208,E2 -1542.208} C_VEL
LIN {X 0,Y 587.719,Z 272.685,A -85,B 0,C 180,E1 -1543.466,E2 -1543.466} C_VEL
LIN {X 0,Y 587.4,Z 270.457,A -85,B 0,C 180,E1 -1543.512,E2 -1543.512} C_VEL
LIN {X 0,Y 587.556,Z 249.352,A -85,B 0,C 180,E1 -1546.323,E2 -1546.323} C_VEL
LIN {X 0,Y 587.664,Z 227.464,A -85,B 0,C 180,E1 -1549.282,E2 -1549.282} C_VEL
LIN {X 0,Y 587.834,Z 209.467,A -85,B 0,C 180,E1 -1551.751,E2 -1551.751} C_VEL
LIN {X 0,Y 587.79,Z 198.815,A -85,B 0,C 180,E1 -1553.236,E2 -1553.236} C_VEL
LIN {X 0,Y 587.322,Z 196.327,A -85,B 0,C 180,E1 -1553.629,E2 -1553.629} C_VEL
LIN {X 0,Y 587.35,Z 196.326,A -85,B 0,C 180,E1 -1556.274,E2 -1556.274} C_VEL
LIN {X 0,Y 587.332,Z 196.319,A -85,B 0,C 180,E1 -1559.13,E2 -1559.13} C_VEL
LIN {X 0,Y 587.327,Z 196.325,A -85,B 0,C 180,E1 -1561.832,E2 -1561.832} C_VEL
LIN {X 0,Y 587.334,Z 196.323,A -85,B 0,C 180,E1 -1564.345,E2 -1564.345} C_VEL
LIN {X 0,Y 587.329,Z 196.319,A -85,B 0,C 180,E1 -1566.743,E2 -1566.743} C_VEL
LIN {X 0,Y 587.323,Z 196.321,A -85,B 0,C 180,E1 -1569.355,E2 -1569.355} C_VEL
LIN {X 0,Y 587.305,Z 196.328,A -85,B 0,C 180,E1 -1572.104,E2 -1572.104} C_VEL
LIN {X 0,Y 587.283,Z 196.325,A -85,B 0,C 180,E1 -1574.908,E2 -1574.908} C_VEL
LIN {X 0,Y 587.317,Z 196.328,A -85,B 0,C 180,E1 -1577.924,E2 -1577.924} C_VEL
LIN {X 0,Y 587.316,Z 196.321,A -85,B 0,C 180,E1 -1580.638,E2 -1580.638} C_VEL
LIN {X 0,Y 587.315,Z 196.324,A -85,B 0,C 180,E1 -1583.288,E2 -1583.288} C_VEL
LIN {X 0,Y 587.333,Z 196.327,A -85,B 0,C 180,E1 -1585.778,E2 -1585.778} C_VEL
LIN {X 0,Y 587.319,Z 196.322,A -85,B 0,C 180,E1 -1588.23,E2 -1588.23} C_VEL
LIN {X 0,Y 587.332,Z 196.319,A -85,B 0,C 180,E1 -1590.858,E2 -1590.858} C_VEL
LIN {X 0,Y 587.314,Z 196.326,A -85,B 0,C 180,E1 -1593.815,E2 -1593.815} C_VEL
LIN {X 0,Y 587.328,Z 196.32,A -85,B 0,C 180,E1 -1596.741,E2 -1596.741} C_VEL
LIN {X 0,Y 587.301,Z 196.328,A -85,B 0,C 180,E1 -1599.694,E2 -1599.694} C_VEL
LIN {X 0,Y 587.29,Z 196.327,A -85,B 0,C 180,E1 -1601.872,E2 -1601.872} C_VEL
LIN {X 0,Y 587.288,Z 196.325,A -85,B 0,C 180,E1 -1604.024,E2 -1604.024} C_VEL
LIN {X 0,Y 587.298,Z 196.326,A -85,B 0,C 180,E1 -1606.858,E2 -1606.858} C_VEL
LIN {X 0,Y 587.352,Z 196.321,A -85,B 0,C 180,E1 -1608.962,E2 -1608.962} C_VEL
LIN {X 0,Y 587.318,Z 196.323,A -85,B 0,C 180,E1 -1611.744,E2 -1611.744} C_VEL
LIN {X 0,Y 587.277,Z 196.327,A -85,B 0,C 180,E1 -1613.817,E2 -1613.817} C_VEL
LIN {X 0,Y 587.258,Z 196.328,A -85,B 0,C 180,E1 -1615.882,E2 -1615.882} C_VEL
LIN {X 0,Y 587.303,Z 196.322,A -85,B 0,C 180,E1 -1617.942,E2 -1617.942} C_VEL
LIN {X 0,Y 587.349,Z 196.32,A -85,B 0,C 180,E1 -1620.685,E2 -1620.685} C_VEL
LIN {X 0,Y 587.296,Z 196.327,A -85,B 0,C 180,E1 -1623.43,E2 -1623.43} C_VEL
LIN {X 0,Y 587.311,Z 196.324,A -85,B 0,C 180,E1 -1625.493,E2 -1625.493} C_VEL
LIN {X 0,Y 587.309,Z 196.322,A -85,B 0,C 180,E1 -1628.256,E2 -1628.256} C_VEL
LIN {X 0,Y 587.369,Z 196.319,A -85,B 0,C 180,E1 -1631.176,E2 -1631.176} C_VEL
LIN {X 0,Y 587.304,Z 196.324,A -85,B 0,C 180,E1 -1634.262,E2 -1634.262} C_VEL
LIN {X 0,Y 587.304,Z 196.323,A -85,B 0,C 180,E1 -1637.407,E2 -1637.407} C_VEL
LIN {X 0,Y 587.28,Z 196.327,A -85,B 0,C 180,E1 -1638.34,E2 -1638.34} C_VEL
LIN {X 0,Y 586.634,Z 196.414,A -85,B 0,C 180,E1 -1638.913,E2 -1638.913} C_VEL
LIN {X 0,Y 583.795,Z 196.767,A -85,B 0,C 180,E1 -1639.841,E2 -1639.841} C_VEL
LIN {X 0,Y 581.377,Z 197.068,A -85,B 0,C 180,E1 -1640.588,E2 -1640.588} C_VEL
LIN {X 0,Y 580.326,Z 197.195,A -85,B 0,C 180,E1 -1641.164,E2 -1641.164} C_VEL
LIN {X 0,Y 580.234,Z 197.204,A -85,B 0,C 180,E1 -1641.36,E2 -1641.36} C_VEL
LIN {X 0,Y 580.249,Z 197.201,A -85,B 0,C 180,E1 -1643.559,E2 -1643.559} C_VEL
LIN {X 0,Y 580.275,Z 197.203,A -85,B 0,C 180,E1 -1646.344,E2 -1646.344} C_VEL
LIN {X 0,Y 580.255,Z 197.204,A -85,B 0,C 180,E1 -1648.978,E2 -1648.978} C_VEL
LIN {X 0,Y 580.266,Z 197.201,A -85,B 0,C 180,E1 -1652.036,E2 -1652.036} C_VEL
LIN {X 0,Y 580.257,Z 197.206,A -85,B 0,C 180,E1 -1654.698,E2 -1654.698} C_VEL
LIN {X 0,Y 580.257,Z 197.2,A -85,B 0,C 180,E1 -1657.271,E2 -1657.271} C_VEL
LIN {X 0,Y 580.26,Z 197.208,A -85,B 0,C 180,E1 -1660.275,E2 -1660.275} C_VEL
LIN {X 0,Y 580.26,Z 197.204,A -85,B 0,C 180,E1 -1662.708,E2 -1662.708} C_VEL
LIN {X 0,Y 580.226,Z 197.205,A -85,B 0,C 180,E1 -1665.613,E2 -1665.613} C_VEL
LIN {X 0,Y 580.282,Z 197.207,A -85,B 0,C 180,E1 -1668.238,E2 -1668.238} C_VEL
LIN {X 0,Y 580.255,Z 197.201,A -85,B 0,C 180,E1 -1670.969,E2 -1670.969} C_VEL
LIN {X 0,Y 580.265,Z 197.201,A -85,B 0,C 180,E1 -1673.601,E2 -1673.601} C_VEL
LIN {X 0,Y 580.281,Z 197.199,A -85,B 0,C 180,E1 -1676.687,E2 -1676.687} C_VEL
LIN {X 0,Y 580.28,Z 197.198,A -85,B 0,C 180,E1 -1679.429,E2 -1679.429} C_VEL
LIN {X 0,Y 580.279,Z 197.205,A -85,B 0,C 180,E1 -1682.145,E2 -1682.145} C_VEL
LIN {X 0,Y 580.307,Z 197.195,A -85,B 0,C 180,E1 -1685.273,E2 -1685.273} C_VEL
LIN {X 0,Y 580.256,Z 197.21,A -85,B 0,C 180,E1 -1687.95,E2 -1687.95} C_VEL
LIN {X 0,Y 580.275,Z 197.198,A -85,B 0,C 180,E1 -1690.916,E2 -1690.916} C_VEL
LIN {X 0,Y 580.249,Z 197.211,A -85,B 0,C 180,E1 -1693.827,E2 -1693.827} C_VEL
LIN {X 0,Y 580.306,Z 197.2,A -85,B 0,C 180,E1 -1695.985,E2 -1695.985} C_VEL
LIN {X 0,Y 580.3,Z 197.195,A -85,B 0,C 180,E1 -1698.829,E2 -1698.829} C_VEL
LIN {X 0,Y 580.321,Z 197.202,A -85,B 0,C 180,E1 -1701.646,E2 -1701.646} C_VEL
LIN {X 0,Y 580.31,Z 197.195,A -85,B 0,C 180,E1 -1704.442,E2 -1704.442} C_VEL
LIN {X 0,Y 580.286,Z 197.309,A -85,B 0,C 180,E1 -1706.725,E2 -1706.725} C_VEL
LIN {X 0,Y 580.402,Z 207.452,A -85,B 0,C 180,E1 -1708.614,E2 -1708.614} C_VEL
LIN {X 0,Y 580.284,Z 222.583,A -85,B 0,C 180,E1 -1711.389,E2 -1711.389} C_VEL
LIN {X 0,Y 580.956,Z 227.052,A -85,B 0,C 180,E1 -1711.474,E2 -1711.474} C_VEL
LIN {X 0,Y 580.763,Z 329.024,A -85,B 0,C 180,E1 -1712.754,E2 -1712.754} C_VEL
LIN {X 0,Y 580.7,Z 342.096,A -85,B 0,C 180,E1 -1713.058,E2 -1713.058} C_VEL
LIN {X 0,Y 580.638,Z 355.21,A -85,B 0,C 180,E1 -1713.514,E2 -1713.514} C_VEL
LIN {X 0,Y 580.527,Z 367.103,A -85,B 0,C 180,E1 -1714.079,E2 -1714.079} C_VEL
LIN {X 0,Y 580.388,Z 378.494,A -85,B 0,C 180,E1 -1714.776,E2 -1714.776} C_VEL
LIN {X 0,Y 580.361,Z 388.745,A -85,B 0,C 180,E1 -1715.56,E2 -1715.56} C_VEL
LIN {X 0,Y 580.301,Z 398.604,A -85,B 0,C 180,E1 -1716.493,E2 -1716.493} C_VEL
LIN {X 0,Y 580.199,Z 407.068,A -85,B 0,C 180,E1 -1717.483,E2 -1717.483} C_VEL
LIN {X 0,Y 580.159,Z 414.364,A -85,B 0,C 180,E1 -1718.534,E2 -1718.534} C_VEL
LIN {X 0,Y 580.133,Z 419.315,A -85,B 0,C 180,E1 -1719.413,E2 -1719.413} C_VEL
LIN {X 0,Y 580.1,Z 424.136,A -85,B 0,C 180,E1 -1720.471,E2 -1720.471} C_VEL
LIN {X 0,Y 580.07,Z 427.837,A -85,B 0,C 180,E1 -1721.532,E2 -1721.532} C_VEL
LIN {X 0,Y 580.05,Z 430.506,A -85,B 0,C 180,E1 -1722.597,E2 -1722.597} C_VEL
LIN {X 0,Y 580.059,Z 431.753,A -85,B 0,C 180,E1 -1723.309,E2 -1723.309} C_VEL
LIN {X 0,Y 580.047,Z 432.707,A -85,B 0,C 180,E1 -1724.235,E2 -1724.235} C_VEL
LIN {X 0,Y 580.018,Z 432.912,A -85,B 0,C 180,E1 -1725.46,E2 -1725.46} C_VEL
LIN {X 0,Y 580.035,Z 432.468,A -85,B 0,C 180,E1 -1726.181,E2 -1726.181} C_VEL
LIN {X 0,Y 580.035,Z 431.556,A -85,B 0,C 180,E1 -1726.905,E2 -1726.905} C_VEL
LIN {X 0,Y 580.046,Z 430.216,A -85,B 0,C 180,E1 -1727.632,E2 -1727.632} C_VEL
LIN {X 0,Y 580.066,Z 427.335,A -85,B 0,C 180,E1 -1728.722,E2 -1728.722} C_VEL
LIN {X 0,Y 580.102,Z 423.28,A -85,B 0,C 180,E1 -1729.829,E2 -1729.829} C_VEL
LIN {X 0,Y 580.105,Z 418.436,A -85,B 0,C 180,E1 -1730.846,E2 -1730.846} C_VEL
LIN {X 0,Y 580.159,Z 412.357,A -85,B 0,C 180,E1 -1731.869,E2 -1731.869} C_VEL
LIN {X 0,Y 580.205,Z 405.533,A -85,B 0,C 180,E1 -1732.805,E2 -1732.805} C_VEL
LIN {X 0,Y 580.273,Z 397.174,A -85,B 0,C 180,E1 -1733.747,E2 -1733.747} C_VEL
LIN {X 0,Y 580.374,Z 387.153,A -85,B 0,C 180,E1 -1734.662,E2 -1734.662} C_VEL
LIN {X 0,Y 580.446,Z 376.4,A -85,B 0,C 180,E1 -1735.456,E2 -1735.456} C_VEL
LIN {X 0,Y 580.571,Z 364.31,A -85,B 0,C 180,E1 -1736.156,E2 -1736.156} C_VEL
LIN {X 0,Y 580.64,Z 352.034,A -85,B 0,C 180,E1 -1736.701,E2 -1736.701} C_VEL
LIN {X 0,Y 580.7,Z 339.344,A -85,B 0,C 180,E1 -1737.111,E2 -1737.111} C_VEL
LIN {X 0,Y 580.731,Z 326.457,A -85,B 0,C 180,E1 -1737.378,E2 -1737.378} C_VEL
LIN {X 0,Y 580.916,Z 226.56,A -85,B 0,C 180,E1 -1738.623,E2 -1738.623} C_VEL
LIN {X 0,Y 580.275,Z 222.588,A -85,B 0,C 180,E1 -1738.7,E2 -1738.7} C_VEL
LIN {X 0,Y 580.399,Z 207.994,A -85,B 0,C 180,E1 -1741.376,E2 -1741.376} C_VEL
LIN {X 0,Y 580.342,Z 197.193,A -85,B 0,C 180,E1 -1743.407,E2 -1743.407} C_VEL
LIN {X 0,Y 580.286,Z 197.207,A -85,B 0,C 180,E1 -1746.4,E2 -1746.4} C_VEL
LIN {X 0,Y 580.296,Z 197.196,A -85,B 0,C 180,E1 -1749.186,E2 -1749.186} C_VEL
LIN {X 0,Y 580.305,Z 197.196,A -85,B 0,C 180,E1 -1751.763,E2 -1751.763} C_VEL
LIN {X 0,Y 580.25,Z 197.205,A -85,B 0,C 180,E1 -1754.624,E2 -1754.624} C_VEL
LIN {X 0,Y 580.291,Z 197.198,A -85,B 0,C 180,E1 -1757.624,E2 -1757.624} C_VEL
LIN {X 0,Y 580.282,Z 197.206,A -85,B 0,C 180,E1 -1760.067,E2 -1760.067} C_VEL
LIN {X 0,Y 580.279,Z 197.197,A -85,B 0,C 180,E1 -1763.063,E2 -1763.063} C_VEL
LIN {X 0,Y 580.284,Z 197.198,A -85,B 0,C 180,E1 -1765.438,E2 -1765.438} C_VEL
LIN {X 0,Y 580.288,Z 197.205,A -85,B 0,C 180,E1 -1767.965,E2 -1767.965} C_VEL
LIN {X 0,Y 580.285,Z 197.196,A -85,B 0,C 180,E1 -1770.686,E2 -1770.686} C_VEL
LIN {X 0,Y 580.3,Z 197.202,A -85,B 0,C 180,E1 -1773.657,E2 -1773.657} C_VEL
LIN {X 0,Y 580.28,Z 197.198,A -85,B 0,C 180,E1 -1776.442,E2 -1776.442} C_VEL
LIN {X 0,Y 580.266,Z 197.204,A -85,B 0,C 180,E1 -1779.437,E2 -1779.437} C_VEL
LIN {X 0,Y 580.263,Z 197.209,A -85,B 0,C 180,E1 -1781.645,E2 -1781.645} C_VEL
LIN {X 0,Y 580.267,Z 197.205,A -85,B 0,C 180,E1 -1783.825,E2 -1783.825} C_VEL
LIN {X 0,Y 580.253,Z 197.2,A -85,B 0,C 180,E1 -1786.696,E2 -1786.696} C_VEL
LIN {X 0,Y 580.279,Z 197.207,A -85,B 0,C 180,E1 -1789.533,E2 -1789.533} C_VEL
LIN {X 0,Y 580.304,Z 197.193,A -85,B 0,C 180,E1 -1792.345,E2 -1792.345} C_VEL
LIN {X 0,Y 580.32,Z 197.198,A -85,B 0,C 180,E1 -1795.137,E2 -1795.137} C_VEL
LIN {X 0,Y 580.294,Z 197.196,A -85,B 0,C 180,E1 -1797.918,E2 -1797.918} C_VEL
LIN {X 0,Y 580.303,Z 197.194,A -85,B 0,C 180,E1 -1800,E2 -1800} C_VEL
LIN {X 0,Y 580.311,Z 197.196,A -85,B 0,C 180,E1 -1802.777,E2 -1802.777} C_VEL
LIN {X 0,Y 580.294,Z 197.197,A -85,B 0,C 180,E1 -1805.56,E2 -1805.56} C_VEL
LIN {X 0,Y 580.268,Z 197.199,A -85,B 0,C 180,E1 -1808.357,E2 -1808.357} C_VEL
LIN {X 0,Y 580.328,Z 197.197,A -85,B 0,C 180,E1 -1811.225,E2 -1811.225} C_VEL
LIN {X 0,Y 580.271,Z 197.199,A -85,B 0,C 180,E1 -1814.337,E2 -1814.337} C_VEL
LIN {X 0,Y 580.277,Z 197.207,A -85,B 0,C 180,E1 -1816.915,E2 -1816.915} C_VEL
LIN {X 0,Y 580.251,Z 197.2,A -85,B 0,C 180,E1 -1819.824,E2 -1819.824} C_VEL
LIN {X 0,Y 580.233,Z 197.204,A -85,B 0,C 180,E1 -1822.054,E2 -1822.054} C_VEL
LIN {X 0,Y 580.248,Z 197.205,A -85,B 0,C 180,E1 -1825.083,E2 -1825.083} C_VEL
LIN {X 0,Y 580.229,Z 197.203,A -85,B 0,C 180,E1 -1827.853,E2 -1827.853} C_VEL
LIN {X 0,Y 580.256,Z 197.21,A -85,B 0,C 180,E1 -1830.577,E2 -1830.577} C_VEL
LIN {X 0,Y 580.255,Z 197.201,A -85,B 0,C 180,E1 -1833.315,E2 -1833.315} C_VEL
LIN {X 0,Y 580.219,Z 197.206,A -85,B 0,C 180,E1 -1835.758,E2 -1835.758} C_VEL
LIN {X 0,Y 580.261,Z 197.205,A -85,B 0,C 180,E1 -1838.149,E2 -1838.149} C_VEL
LIN {X 0,Y 580.277,Z 197.199,A -85,B 0,C 180,E1 -1840.846,E2 -1840.846} C_VEL
LIN {X 0,Y 580.253,Z 197.202,A -85,B 0,C 180,E1 -1843.661,E2 -1843.661} C_VEL
LIN {X 0,Y 580.249,Z 197.205,A -85,B 0,C 180,E1 -1846.613,E2 -1846.613} C_VEL
LIN {X 0,Y 580.28,Z 197.197,A -85,B 0,C 180,E1 -1849.158,E2 -1849.158} C_VEL
LIN {X 0,Y 580.275,Z 197.205,A -85,B 0,C 180,E1 -1851.929,E2 -1851.929} C_VEL
LIN {X 0,Y 580.272,Z 197.203,A -85,B 0,C 180,E1 -1854.456,E2 -1854.456} C_VEL
LIN {X 0,Y 580.28,Z 197.198,A -85,B 0,C 180,E1 -1856.976,E2 -1856.976} C_VEL
LIN {X 0,Y 580.287,Z 197.199,A -85,B 0,C 180,E1 -1859.426,E2 -1859.426} C_VEL
LIN {X 0,Y 580.254,Z 197.208,A -85,B 0,C 180,E1 -1862.15,E2 -1862.15} C_VEL
LIN {X 0,Y 580.301,Z 197.197,A -85,B 0,C 180,E1 -1864.921,E2 -1864.921} C_VEL
LIN {X 0,Y 580.312,Z 197.38,A -85,B 0,C 180,E1 -1866.302,E2 -1866.302} C_VEL
LIN {X 0,Y 580.948,Z 201.945,A -85,B 0,C 180,E1 -1866.956,E2 -1866.956} C_VEL
LIN {X 0,Y 580.837,Z 221.414,A -85,B 0,C 180,E1 -1869.644,E2 -1869.644} C_VEL
LIN {X 0,Y 580.587,Z 242.819,A -85,B 0,C 180,E1 -1872.585,E2 -1872.585} C_VEL
LIN {X 0,Y 580.465,Z 262.628,A -85,B 0,C 180,E1 -1875.271,E2 -1875.271} C_VEL
LIN {X 0,Y 580.413,Z 270.522,A -85,B 0,C 180,E1 -1876.331,E2 -1876.331} C_VEL
LIN {X 0,Y 580.96,Z 276.511,A -85,B 0,C 180,E1 -1876.422,E2 -1876.422} C_VEL
LIN {X 0,Y 580.802,Z 378.942,A -85,B 0,C 180,E1 -1877.708,E2 -1877.708} C_VEL
LIN {X 0,Y 580.74,Z 392.215,A -85,B 0,C 180,E1 -1878.017,E2 -1878.017} C_VEL
LIN {X 0,Y 580.656,Z 405.145,A -85,B 0,C 180,E1 -1878.467,E2 -1878.467} C_VEL
LIN {X 0,Y 580.553,Z 416.625,A -85,B 0,C 180,E1 -1879.008,E2 -1879.008} C_VEL
LIN {X 0,Y 580.445,Z 428.198,A -85,B 0,C 180,E1 -1879.712,E2 -1879.712} C_VEL
LIN {X 0,Y 580.345,Z 438.596,A -85,B 0,C 180,E1 -1880.502,E2 -1880.502} C_VEL
LIN {X 0,Y 580.272,Z 447.108,A -85,B 0,C 180,E1 -1881.292,E2 -1881.292} C_VEL
LIN {X 0,Y 580.222,Z 454.956,A -85,B 0,C 180,E1 -1882.168,E2 -1882.168} C_VEL
LIN {X 0,Y 580.154,Z 462.648,A -85,B 0,C 180,E1 -1883.221,E2 -1883.221} C_VEL
LIN {X 0,Y 580.139,Z 469.676,A -85,B 0,C 180,E1 -1884.438,E2 -1884.438} C_VEL
LIN {X 0,Y 580.108,Z 474.369,A -85,B 0,C 180,E1 -1885.483,E2 -1885.483} C_VEL
LIN {X 0,Y 580.123,Z 477.954,A -85,B 0,C 180,E1 -1886.526,E2 -1886.526} C_VEL
LIN {X 0,Y 580.043,Z 479.806,A -85,B 0,C 180,E1 -1887.221,E2 -1887.221} C_VEL
LIN {X 0,Y 580.04,Z 481.197,A -85,B 0,C 180,E1 -1887.916,E2 -1887.916} C_VEL
LIN {X 0,Y 580.04,Z 482.784,A -85,B 0,C 180,E1 -1889.305,E2 -1889.305} C_VEL
LIN {X 0,Y 580.037,Z 483,A -85,B 0,C 180,E1 -1889.999,E2 -1889.999} C_VEL
LIN {X 0,Y 580.046,Z 482.188,A -85,B 0,C 180,E1 -1891.387,E2 -1891.387} C_VEL
LIN {X 0,Y 580.04,Z 481.202,A -85,B 0,C 180,E1 -1892.082,E2 -1892.082} C_VEL
LIN {X 0,Y 580.043,Z 479.813,A -85,B 0,C 180,E1 -1892.776,E2 -1892.776} C_VEL
LIN {X 0,Y 580.109,Z 476.901,A -85,B 0,C 180,E1 -1893.819,E2 -1893.819} C_VEL
LIN {X 0,Y 580.053,Z 472.956,A -85,B 0,C 180,E1 -1894.864,E2 -1894.864} C_VEL
LIN {X 0,Y 580.166,Z 467.876,A -85,B 0,C 180,E1 -1895.908,E2 -1895.908} C_VEL
LIN {X 0,Y 580.157,Z 461.482,A -85,B 0,C 180,E1 -1896.956,E2 -1896.956} C_VEL
LIN {X 0,Y 580.241,Z 453.495,A -85,B 0,C 180,E1 -1898.005,E2 -1898.005} C_VEL
LIN {X 0,Y 580.304,Z 445.357,A -85,B 0,C 180,E1 -1898.881,E2 -1898.881} C_VEL
LIN {X 0,Y 580.372,Z 435.427,A -85,B 0,C 180,E1 -1899.759,E2 -1899.759} C_VEL
LIN {X 0,Y 580.494,Z 424.21,A -85,B 0,C 180,E1 -1900.549,E2 -1900.549} C_VEL
LIN {X 0,Y 580.604,Z 413.223,A -85,B 0,C 180,E1 -1901.165,E2 -1901.165} C_VEL
LIN {X 0,Y 580.654,Z 401.044,A -85,B 0,C 180,E1 -1901.694,E2 -1901.694} C_VEL
LIN {X 0,Y 580.732,Z 388.274,A -85,B 0,C 180,E1 -1902.092,E2 -1902.092} C_VEL
LIN {X 0,Y 580.829,Z 374.763,A -85,B 0,C 180,E1 -1902.356,E2 -1902.356} C_VEL
LIN {X 0,Y 580.802,Z 273.357,A -85,B 0,C 180,E1 -1903.621,E2 -1903.621} C_VEL
LIN {X 0,Y 580.406,Z 270.457,A -85,B 0,C 180,E1 -1903.677,E2 -1903.677} C_VEL
LIN {X 0,Y 580.594,Z 248.022,A -85,B 0,C 180,E1 -1906.705,E2 -1906.705} C_VEL
LIN {X 0,Y 580.776,Z 226.609,A -85,B 0,C 180,E1 -1909.638,E2 -1909.638} C_VEL
LIN {X 0,Y 580.939,Z 206.666,A -85,B 0,C 180,E1 -1912.397,E2 -1912.397} C_VEL
LIN {X 0,Y 580.858,Z 200.237,A -85,B 0,C 180,E1 -1913.288,E2 -1913.288} C_VEL
LIN {X 0,Y 580.275,Z 197.206,A -85,B 0,C 180,E1 -1913.744,E2 -1913.744} C_VEL
LIN {X 0,Y 580.293,Z 197.2,A -85,B 0,C 180,E1 -1916.619,E2 -1916.619} C_VEL
LIN {X 0,Y 580.287,Z 197.197,A -85,B 0,C 180,E1 -1919.306,E2 -1919.306} C_VEL
LIN {X 0,Y 580.279,Z 197.205,A -85,B 0,C 180,E1 -1922.197,E2 -1922.197} C_VEL
LIN {X 0,Y 580.279,Z 197.198,A -85,B 0,C 180,E1 -1924.692,E2 -1924.692} C_VEL
LIN {X 0,Y 580.277,Z 197.198,A -85,B 0,C 180,E1 -1927.265,E2 -1927.265} C_VEL
LIN {X 0,Y 580.273,Z 197.202,A -85,B 0,C 180,E1 -1930.268,E2 -1930.268} C_VEL
LIN {X 0,Y 580.25,Z 197.201,A -85,B 0,C 180,E1 -1932.702,E2 -1932.702} C_VEL
LIN {X 0,Y 580.241,Z 197.208,A -85,B 0,C 180,E1 -1935.605,E2 -1935.605} C_VEL
LIN {X 0,Y 580.285,Z 197.2,A -85,B 0,C 180,E1 -1938.231,E2 -1938.231} C_VEL
LIN {X 0,Y 580.256,Z 197.2,A -85,B 0,C 180,E1 -1940.963,E2 -1940.963} C_VEL
LIN {X 0,Y 580.258,Z 197.208,A -85,B 0,C 180,E1 -1943.595,E2 -1943.595} C_VEL
LIN {X 0,Y 580.283,Z 197.199,A -85,B 0,C 180,E1 -1946.143,E2 -1946.143} C_VEL
LIN {X 0,Y 580.251,Z 197.2,A -85,B 0,C 180,E1 -1948.613,E2 -1948.613} C_VEL
LIN {X 0,Y 580.277,Z 197.2,A -85,B 0,C 180,E1 -1951.023,E2 -1951.023} C_VEL
LIN {X 0,Y 580.281,Z 197.205,A -85,B 0,C 180,E1 -1953.655,E2 -1953.655} C_VEL
LIN {X 0,Y 580.259,Z 197.2,A -85,B 0,C 180,E1 -1956.441,E2 -1956.441} C_VEL
LIN {X 0,Y 580.25,Z 197.211,A -85,B 0,C 180,E1 -1959.436,E2 -1959.436} C_VEL
LIN {X 0,Y 580.246,Z 197.207,A -85,B 0,C 180,E1 -1961.644,E2 -1961.644} C_VEL
LIN {X 0,Y 580.245,Z 197.204,A -85,B 0,C 180,E1 -1963.824,E2 -1963.824} C_VEL
LIN {X 0,Y 580.249,Z 197.202,A -85,B 0,C 180,E1 -1966.695,E2 -1966.695} C_VEL
LIN {X 0,Y 580.271,Z 197.204,A -85,B 0,C 180,E1 -1969.533,E2 -1969.533} C_VEL
LIN {X 0,Y 580.284,Z 197.197,A -85,B 0,C 180,E1 -1972.344,E2 -1972.344} C_VEL
LIN {X 0,Y 580.298,Z 197.205,A -85,B 0,C 180,E1 -1975.137,E2 -1975.137} C_VEL
LIN {X 0,Y 580.275,Z 197.198,A -85,B 0,C 180,E1 -1977.918,E2 -1977.918} C_VEL
LIN {X 0,Y 580.318,Z 197.196,A -85,B 0,C 180,E1 -1980.694,E2 -1980.694} C_VEL
LIN {X 0,Y 580.245,Z 197.204,A -85,B 0,C 180,E1 -1983.472,E2 -1983.472} C_VEL
LIN {X 0,Y 580.274,Z 197.199,A -85,B 0,C 180,E1 -1985.56,E2 -1985.56} C_VEL
LIN {X 0,Y 580.275,Z 197.199,A -85,B 0,C 180,E1 -1988.357,E2 -1988.357} C_VEL
LIN {X 0,Y 580.322,Z 197.196,A -85,B 0,C 180,E1 -1991.234,E2 -1991.234} C_VEL
LIN {X 0,Y 580.255,Z 197.203,A -85,B 0,C 180,E1 -1994.34,E2 -1994.34} C_VEL
LIN {X 0,Y 580.286,Z 197.204,A -85,B 0,C 180,E1 -1996.926,E2 -1996.926} C_VEL
LIN {X 0,Y 580.259,Z 197.2,A -85,B 0,C 180,E1 -1999.824,E2 -1999.824} C_VEL
LIN {X 0,Y 580.234,Z 197.204,A -85,B 0,C 180,E1 -2001.36,E2 -2001.36} C_VEL
LIN {X 0,Y 579.545,Z 197.29,A -85,B 0,C 180,E1 -2001.939,E2 -2001.939} C_VEL
LIN {X 0,Y 576.673,Z 197.653,A -85,B 0,C 180,E1 -2002.879,E2 -2002.879} C_VEL
LIN {X 0,Y 574.275,Z 197.948,A -85,B 0,C 180,E1 -2003.636,E2 -2003.636} C_VEL
LIN {X 0,Y 573.271,Z 198.074,A -85,B 0,C 180,E1 -2004.22,E2 -2004.22} C_VEL
LIN {X 0,Y 573.202,Z 198.085,A -85,B 0,C 180,E1 -2004.418,E2 -2004.418} C_VEL
LIN {X 0,Y 573.214,Z 198.081,A -85,B 0,C 180,E1 -2006.978,E2 -2006.978} C_VEL
LIN {X 0,Y 573.202,Z 198.079,A -85,B 0,C 180,E1 -2009.492,E2 -2009.492} C_VEL
LIN {X 0,Y 573.212,Z 198.085,A -85,B 0,C 180,E1 -2012.647,E2 -2012.647} C_VEL
LIN {X 0,Y 573.224,Z 198.077,A -85,B 0,C 180,E1 -2015.186,E2 -2015.186} C_VEL
LIN {X 0,Y 573.194,Z 198.081,A -85,B 0,C 180,E1 -2017.811,E2 -2017.811} C_VEL
LIN {X 0,Y 573.23,Z 198.083,A -85,B 0,C 180,E1 -2020.531,E2 -2020.531} C_VEL
LIN {X 0,Y 573.21,Z 198.078,A -85,B 0,C 180,E1 -2023.362,E2 -2023.362} C_VEL
LIN {X 0,Y 573.209,Z 198.082,A -85,B 0,C 180,E1 -2026.645,E2 -2026.645} C_VEL
LIN {X 0,Y 573.228,Z 198.076,A -85,B 0,C 180,E1 -2029.48,E2 -2029.48} C_VEL
LIN {X 0,Y 573.207,Z 198.088,A -85,B 0,C 180,E1 -2032.196,E2 -2032.196} C_VEL
LIN {X 0,Y 573.229,Z 198.076,A -85,B 0,C 180,E1 -2034.819,E2 -2034.819} C_VEL
LIN {X 0,Y 573.23,Z 198.076,A -85,B 0,C 180,E1 -2037.358,E2 -2037.358} C_VEL
LIN {X 0,Y 573.23,Z 198.078,A -85,B 0,C 180,E1 -2040.515,E2 -2040.515} C_VEL
LIN {X 0,Y 573.202,Z 198.079,A -85,B 0,C 180,E1 -2043.026,E2 -2043.026} C_VEL
LIN {X 0,Y 573.26,Z 198.073,A -85,B 0,C 180,E1 -2045.369,E2 -2045.369} C_VEL
LIN {X 0,Y 573.215,Z 198.079,A -85,B 0,C 180,E1 -2048.422,E2 -2048.422} C_VEL
LIN {X 0,Y 573.258,Z 198.072,A -85,B 0,C 180,E1 -2050.734,E2 -2050.734} C_VEL
LIN {X 0,Y 573.221,Z 198.083,A -85,B 0,C 180,E1 -2053.624,E2 -2053.624} C_VEL
LIN {X 0,Y 573.251,Z 198.083,A -85,B 0,C 180,E1 -2055.809,E2 -2055.809} C_VEL
LIN {X 0,Y 573.258,Z 198.072,A -85,B 0,C 180,E1 -2058.747,E2 -2058.747} C_VEL
LIN {X 0,Y 573.276,Z 198.077,A -85,B 0,C 180,E1 -2061.542,E2 -2061.542} C_VEL
LIN {X 0,Y 573.279,Z 198.071,A -85,B 0,C 180,E1 -2064.373,E2 -2064.373} C_VEL
LIN {X 0,Y 573.237,Z 198.208,A -85,B 0,C 180,E1 -2066.663,E2 -2066.663} C_VEL
LIN {X 0,Y 573.411,Z 206.587,A -85,B 0,C 180,E1 -2068.245,E2 -2068.245} C_VEL
LIN {X 0,Y 573.242,Z 221.701,A -85,B 0,C 180,E1 -2071.055,E2 -2071.055} C_VEL
LIN {X 0,Y 573.243,Z 222.65,A -85,B 0,C 180,E1 -2071.23,E2 -2071.23} C_VEL
LIN {X 0,Y 574.069,Z 227.708,A -85,B 0,C 180,E1 -2071.316,E2 -2071.316} C_VEL
LIN {X 0,Y 573.847,Z 329.437,A -85,B 0,C 180,E1 -2072.611,E2 -2072.611} C_VEL
LIN {X 0,Y 573.764,Z 342.381,A -85,B 0,C 180,E1 -2072.919,E2 -2072.919} C_VEL
LIN {X 0,Y 573.679,Z 355.428,A -85,B 0,C 180,E1 -2073.381,E2 -2073.381} C_VEL
LIN {X 0,Y 573.537,Z 367.263,A -85,B 0,C 180,E1 -2073.953,E2 -2073.953} C_VEL
LIN {X 0,Y 573.376,Z 378.627,A -85,B 0,C 180,E1 -2074.659,E2 -2074.659} C_VEL
LIN {X 0,Y 573.331,Z 388.858,A -85,B 0,C 180,E1 -2075.452,E2 -2075.452} C_VEL
LIN {X 0,Y 573.241,Z 398.13,A -85,B 0,C 180,E1 -2076.336,E2 -2076.336} C_VEL
LIN {X 0,Y 573.128,Z 407.14,A -85,B 0,C 180,E1 -2077.398,E2 -2077.398} C_VEL
LIN {X 0,Y 573.082,Z 414.422,A -85,B 0,C 180,E1 -2078.463,E2 -2078.463} C_VEL
LIN {X 0,Y 573.031,Z 420.273,A -85,B 0,C 180,E1 -2079.531,E2 -2079.531} C_VEL
LIN {X 0,Y 573.023,Z 424.884,A -85,B 0,C 180,E1 -2080.601,E2 -2080.601} C_VEL
LIN {X 0,Y 572.979,Z 427.323,A -85,B 0,C 180,E1 -2081.318,E2 -2081.318} C_VEL
LIN {X 0,Y 572.951,Z 429.32,A -85,B 0,C 180,E1 -2082.036,E2 -2082.036} C_VEL
LIN {X 0,Y 572.946,Z 430.891,A -85,B 0,C 180,E1 -2082.756,E2 -2082.756} C_VEL
LIN {X 0,Y 572.968,Z 432.001,A -85,B 0,C 180,E1 -2083.477,E2 -2083.477} C_VEL
LIN {X 0,Y 572.959,Z 432.757,A -85,B 0,C 180,E1 -2084.299,E2 -2084.299} C_VEL
LIN {X 0,Y 572.915,Z 432.846,A -85,B 0,C 180,E1 -2085.657,E2 -2085.657} C_VEL
LIN {X 0,Y 572.936,Z 431.594,A -85,B 0,C 180,E1 -2086.904,E2 -2086.904} C_VEL
LIN {X 0,Y 572.953,Z 429.808,A -85,B 0,C 180,E1 -2087.857,E2 -2087.857} C_VEL
LIN {X 0,Y 572.968,Z 425.969,A -85,B 0,C 180,E1 -2089.183,E2 -2089.183} C_VEL
LIN {X 0,Y 573.012,Z 420.742,A -85,B 0,C 180,E1 -2090.459,E2 -2090.459} C_VEL
LIN {X 0,Y 573.089,Z 414.683,A -85,B 0,C 180,E1 -2091.585,E2 -2091.585} C_VEL
LIN {X 0,Y 573.133,Z 406.913,A -85,B 0,C 180,E1 -2092.721,E2 -2092.721} C_VEL
LIN {X 0,Y 573.227,Z 398.881,A -85,B 0,C 180,E1 -2093.673,E2 -2093.673} C_VEL
LIN {X 0,Y 573.328,Z 388.949,A -85,B 0,C 180,E1 -2094.63,E2 -2094.63} C_VEL
LIN {X 0,Y 573.429,Z 377.652,A -85,B 0,C 180,E1 -2095.498,E2 -2095.498} C_VEL
LIN {X 0,Y 573.578,Z 366.604,A -85,B 0,C 180,E1 -2096.173,E2 -2096.173} C_VEL
LIN {X 0,Y 573.682,Z 354.194,A -85,B 0,C 180,E1 -2096.759,E2 -2096.759} C_VEL
LIN {X 0,Y 573.743,Z 341.135,A -85,B 0,C 180,E1 -2097.208,E2 -2097.208} C_VEL
LIN {X 0,Y 573.805,Z 328.96,A -85,B 0,C 180,E1 -2097.489,E2 -2097.489} C_VEL
LIN {X 0,Y 574.029,Z 227.401,A -85,B 0,C 180,E1 -2098.778,E2 -2098.778} C_VEL
LIN {X 0,Y 573.241,Z 222.563,A -85,B 0,C 180,E1 -2098.876,E2 -2098.876} C_VEL
LIN {X 0,Y 573.363,Z 207.902,A -85,B 0,C 180,E1 -2101.6,E2 -2101.6} C_VEL
LIN {X 0,Y 573.31,Z 198.07,A -85,B 0,C 180,E1 -2103.451,E2 -2103.451} C_VEL
LIN {X 0,Y 573.25,Z 198.078,A -85,B 0,C 180,E1 -2106.047,E2 -2106.047} C_VEL
LIN {X 0,Y 573.237,Z 198.08,A -85,B 0,C 180,E1 -2108.699,E2 -2108.699} C_VEL
LIN {X 0,Y 573.25,Z 198.074,A -85,B 0,C 180,E1 -2111.595,E2 -2111.595} C_VEL
LIN {X 0,Y 573.221,Z 198.086,A -85,B 0,C 180,E1 -2114.331,E2 -2114.331} C_VEL
LIN {X 0,Y 573.241,Z 198.075,A -85,B 0,C 180,E1 -2117.355,E2 -2117.355} C_VEL
LIN {X 0,Y 573.232,Z 198.081,A -85,B 0,C 180,E1 -2120.392,E2 -2120.392} C_VEL
LIN {X 0,Y 573.234,Z 198.075,A -85,B 0,C 180,E1 -2123.076,E2 -2123.076} C_VEL
LIN {X 0,Y 573.253,Z 198.077,A -85,B 0,C 180,E1 -2125.671,E2 -2125.671} C_VEL
LIN {X 0,Y 573.228,Z 198.081,A -85,B 0,C 180,E1 -2128.184,E2 -2128.184} C_VEL
LIN {X 0,Y 573.248,Z 198.073,A -85,B 0,C 180,E1 -2130.633,E2 -2130.633} C_VEL
LIN {X 0,Y 573.243,Z 198.078,A -85,B 0,C 180,E1 -2133.499,E2 -2133.499} C_VEL
LIN {X 0,Y 573.238,Z 198.078,A -85,B 0,C 180,E1 -2136.135,E2 -2136.135} C_VEL
LIN {X 0,Y 573.229,Z 198.074,A -85,B 0,C 180,E1 -2138.705,E2 -2138.705} C_VEL
LIN {X 0,Y 573.221,Z 198.082,A -85,B 0,C 180,E1 -2141.411,E2 -2141.411} C_VEL
LIN {X 0,Y 573.242,Z 198.083,A -85,B 0,C 180,E1 -2143.622,E2 -2143.622} C_VEL
LIN {X 0,Y 573.211,Z 198.077,A -85,B 0,C 180,E1 -2146.529,E2 -2146.529} C_VEL
LIN {X 0,Y 573.25,Z 198.081,A -85,B 0,C 180,E1 -2149.403,E2 -2149.403} C_VEL
LIN {X 0,Y 573.254,Z 198.072,A -85,B 0,C 180,E1 -2152.25,E2 -2152.25} C_VEL
LIN {X 0,Y 573.259,Z 198.072,A -85,B 0,C 180,E1 -2154.372,E2 -2154.372} C_VEL
LIN {X 0,Y 573.286,Z 198.075,A -85,B 0,C 180,E1 -2157.19,E2 -2157.19} C_VEL
LIN {X 0,Y 573.274,Z 198.07,A -85,B 0,C 180,E1 -2160,E2 -2160} C_VEL
LIN {X 0,Y 573.277,Z 198.072,A -85,B 0,C 180,E1 -2162.811,E2 -2162.811} C_VEL
LIN {X 0,Y 573.259,Z 198.073,A -85,B 0,C 180,E1 -2165.629,E2 -2165.629} C_VEL
LIN {X 0,Y 573.234,Z 198.075,A -85,B 0,C 180,E1 -2167.751,E2 -2167.751} C_VEL
LIN {X 0,Y 573.258,Z 198.074,A -85,B 0,C 180,E1 -2170.597,E2 -2170.597} C_VEL
LIN {X 0,Y 573.193,Z 198.081,A -85,B 0,C 180,E1 -2173.472,E2 -2173.472} C_VEL
LIN {X 0,Y 573.197,Z 198.08,A -85,B 0,C 180,E1 -2175.649,E2 -2175.649} C_VEL
LIN {X 0,Y 573.203,Z 198.078,A -85,B 0,C 180,E1 -2177.85,E2 -2177.85} C_VEL
LIN {X 0,Y 573.209,Z 198.078,A -85,B 0,C 180,E1 -2180.078,E2 -2180.078} C_VEL
LIN {X 0,Y 573.198,Z 198.083,A -85,B 0,C 180,E1 -2182.34,E2 -2182.34} C_VEL
LIN {X 0,Y 573.201,Z 198.08,A -85,B 0,C 180,E1 -2185.413,E2 -2185.413} C_VEL
LIN {X 0,Y 573.2,Z 198.088,A -85,B 0,C 180,E1 -2188.567,E2 -2188.567} C_VEL
LIN {X 0,Y 573.192,Z 198.083,A -85,B 0,C 180,E1 -2190.996,E2 -2190.996} C_VEL
LIN {X 0,Y 573.216,Z 198.077,A -85,B 0,C 180,E1 -2193.523,E2 -2193.523} C_VEL
LIN {X 0,Y 573.169,Z 198.087,A -85,B 0,C 180,E1 -2196.055,E2 -2196.055} C_VEL
LIN {X 0,Y 573.213,Z 198.083,A -85,B 0,C 180,E1 -2198.704,E2 -2198.704} C_VEL
LIN {X 0,Y 573.222,Z 198.075,A -85,B 0,C 180,E1 -2201.596,E2 -2201.596} C_VEL
LIN {X 0,Y 573.211,Z 198.087,A -85,B 0,C 180,E1 -2204.336,E2 -2204.336} C_VEL
LIN {X 0,Y 573.207,Z 198.079,A -85,B 0,C 180,E1 -2207.363,E2 -2207.363} C_VEL
LIN {X 0,Y 573.225,Z 198.082,A -85,B 0,C 180,E1 -2210.394,E2 -2210.394} C_VEL
LIN {X 0,Y 573.241,Z 198.073,A -85,B 0,C 180,E1 -2213.079,E2 -2213.079} C_VEL
LIN {X 0,Y 573.255,Z 198.077,A -85,B 0,C 180,E1 -2215.673,E2 -2215.673} C_VEL
LIN {X 0,Y 573.23,Z 198.083,A -85,B 0,C 180,E1 -2218.186,E2 -2218.186} C_VEL
LIN {X 0,Y 573.255,Z 198.074,A -85,B 0,C 180,E1 -2220.635,E2 -2220.635} C_VEL
LIN {X 0,Y 573.251,Z 198.082,A -85,B 0,C 180,E1 -2223.811,E2 -2223.811} C_VEL
LIN {X 0,Y 573.269,Z 198.189,A -85,B 0,C 180,E1 -2226.159,E2 -2226.159} C_VEL
LIN {X 0,Y 574.002,Z 203.539,A -85,B 0,C 180,E1 -2226.934,E2 -2226.934} C_VEL
LIN {X 0,Y 573.853,Z 223.977,A -85,B 0,C 180,E1 -2229.759,E2 -2229.759} C_VEL
LIN {X 0,Y 573.615,Z 245.479,A -85,B 0,C 180,E1 -2232.735,E2 -2232.735} C_VEL
LIN {X 0,Y 573.464,Z 264.929,A -85,B 0,C 180,E1 -2235.401,E2 -2235.401} C_VEL
LIN {X 0,Y 573.417,Z 270.522,A -85,B 0,C 180,E1 -2236.161,E2 -2236.161} C_VEL
LIN {X 0,Y 574.054,Z 276.511,A -85,B 0,C 180,E1 -2236.256,E2 -2236.256} C_VEL
LIN {X 0,Y 573.879,Z 378.942,A -85,B 0,C 180,E1 -2237.557,E2 -2237.557} C_VEL
LIN {X 0,Y 573.798,Z 392.214,A -85,B 0,C 180,E1 -2237.87,E2 -2237.87} C_VEL
LIN {X 0,Y 573.703,Z 404.372,A -85,B 0,C 180,E1 -2238.294,E2 -2238.294} C_VEL
LIN {X 0,Y 573.58,Z 416.623,A -85,B 0,C 180,E1 -2238.873,E2 -2238.873} C_VEL
LIN {X 0,Y 573.436,Z 428.196,A -85,B 0,C 180,E1 -2239.585,E2 -2239.585} C_VEL
LIN {X 0,Y 573.332,Z 438.598,A -85,B 0,C 180,E1 -2240.385,E2 -2240.385} C_VEL
LIN {X 0,Y 573.241,Z 447.109,A -85,B 0,C 180,E1 -2241.184,E2 -2241.184} C_VEL
LIN {X 0,Y 573.161,Z 454.956,A -85,B 0,C 180,E1 -2242.071,E2 -2242.071} C_VEL
LIN {X 0,Y 573.074,Z 462.578,A -85,B 0,C 180,E1 -2243.126,E2 -2243.126} C_VEL
LIN {X 0,Y 573.07,Z 469.676,A -85,B 0,C 180,E1 -2244.369,E2 -2244.369} C_VEL
LIN {X 0,Y 573.029,Z 474.369,A -85,B 0,C 180,E1 -2245.427,E2 -2245.427} C_VEL
LIN {X 0,Y 573.022,Z 477.955,A -85,B 0,C 180,E1 -2246.483,E2 -2246.483} C_VEL
LIN {X 0,Y 572.959,Z 479.806,A -85,B 0,C 180,E1 -2247.187,E2 -2247.187} C_VEL
LIN {X 0,Y 572.94,Z 481.196,A -85,B 0,C 180,E1 -2247.89,E2 -2247.89} C_VEL
LIN {X 0,Y 572.941,Z 482.784,A -85,B 0,C 180,E1 -2249.296,E2 -2249.296} C_VEL
LIN {X 0,Y 572.938,Z 483,A -85,B 0,C 180,E1 -2249.999,E2 -2249.999} C_VEL
LIN {X 0,Y 572.946,Z 482.188,A -85,B 0,C 180,E1 -2251.404,E2 -2251.404} C_VEL
LIN {X 0,Y 572.939,Z 481.201,A -85,B 0,C 180,E1 -2252.108,E2 -2252.108} C_VEL
LIN {X 0,Y 572.959,Z 479.813,A -85,B 0,C 180,E1 -2252.811,E2 -2252.811} C_VEL
LIN {X 0,Y 573.014,Z 476.901,A -85,B 0,C 180,E1 -2253.866,E2 -2253.866} C_VEL
